		parameterCount:= pCurrentObject.getParametersCount();
		IF parameterCount>0 THEN
			FOR parameterIndex:=0 TO parameterCount-1 DO
				curData:=pCurrentObject.getParametrName(parameterIndex);
				SysFileStreamFPutS(File:=h_file,str:=ADR(devisor));
				SysFileStreamFPutS(File:=h_file,str:=ADR(curData));	
			END_FOR
		ELSE
				SysFileStreamFPutS(File:=h_file,str:=ADR(devisor));				
		END_IF			
		currentObject:=currentObject.NextElem;
	UNTIL 	currentObject =0
	END_REPEAT	
END_IF
END_METHOD

METHOD PRIVATE writeDataRow:BOOL
VAR_INPUT
		h_file:RTS_IEC_HANDLE;
		currentSlice:LAT.IElement;
END_VAR
VAR
	curData:STRING;
	currentObject: LAT.IElement;
	pCurrentObject:IObjectListener;	
	pCurrentSlice: POINTER TO TimeSlice;	
	parameterIndex:WORD;
	parameterCount:WORD;
END_VAR
__QUERYPOINTER (currentSlice,pCurrentSlice);
IF NOT pCurrentSlice^.values.ListIsEmpty THEN
	SysFileStreamFPutS(File:=h_file,str:=ADR(endln));
	curData:=timeToString(hrTime:=pCurrentSlice^.timeStamp);
	SysFileStreamFPutS(File:=h_file,str:=ADR(curData));

	currentObject:=pCurrentSlice^.values.HeadElem;
	REPEAT
		__QUERYINTERFACE (currentObject,pCurrentObject);

		parameterCount:= pCurrentObject.getParametersCount();
		IF parameterCount>0 THEN
			FOR parameterIndex:=0 TO parameterCount-1 DO
				curData:=pCurrentObject.getParametrValue(parameterIndex);
				SysFileStreamFPutS(File:=h_file,str:=ADR(devisor));
				SysFileStreamFPutS(File:=h_file,str:=ADR(curData));	
			END_FOR
		ELSE
				SysFileStreamFPutS(File:=h_file,str:=ADR(devisor));				
		END_IF		
		
		currentObject:=currentObject.NextElem;
	UNTIL 	currentObject =0
	END_REPEAT			
END_IF
writeDataRow:=pCurrentSlice^.timeStamp>=lastSavedTimeStamp;
END_METHOD

METHOD PRIVATE countinueDataWrite
VAR_INPUT
END_VAR
VAR
	timeKvant:TON:=(PT:=writeFileTimeKvant);
	isLastRow:BOOL;
END_VAR
timeKvant(IN:=FALSE);
timeKvant(IN:=TRUE);

IF currentWritedSlice=0 THEN
	currentWritedSlice:=TimeSlices.HeadElem;
END_IF;		
REPEAT
	isLastRow:= writeDataRow(archiveFileHandle,currentWritedSlice);
	timeKvant();
	currentWritedSlice:=currentWritedSlice.NextElem;
UNTIL 	(currentWritedSlice=0) OR isLastRow OR  timeKvant.Q
END_REPEAT	

IF isLastRow OR currentWritedSlice=0 THEN
	SysFileStreamFClose(File:=archiveFileHandle);
	archiveFileHandle:=0;
	currentWritedSlice:=0;
END_IF;
END_METHOD

METHOD PUBLIC register
VAR_INPUT
END_VAR
VAR

END_VAR
provider.RegisterArchive(nArchive:=THIS);
END_METHOD

METHOD FB_init : BOOL
VAR_INPUT
  bInitRetains : BOOL; // if TRUE, the retain variables are initialized (warm start / cold start)
  bInCopyCode : BOOL;  // if TRUE, the instance afterwards gets moved into the copy code (online change)
  table: POINTER TO TableDescriptor;
END_VAR
register();
END_METHOD

METHOD PUBLIC startAccident
VAR_INPUT
	descript:STRING;
END_VAR
IF NOT (accidentStarted OR (archiveFileHandle<>0)) THEN
	SysTimeRtcHighResGet(accidentTime);
	accidentStarted:=TRUE;	
	accidentDesc:=descript;
END_IF
END_METHOD

METHOD PUBLIC writeLog
VAR_INPUT
	fileName:STRING;
	append:BOOL;
END_VAR
VAR
	fileMode:STRING;
END_VAR
IF append THEN
	fileMode:='a';
ELSE
	fileMode:='w';		
END_IF
archiveFileHandle:=SysFileStreamFOpen(FileName:=fileName,Mode:=fileMode);

IF archiveFileHandle=0 THEN
	RETURN;
END_IF

IF lastTimeSlice<>0 THEN
	IF NOT append THEN
		writeHead(archiveFileHandle);
	END_IF
	countinueDataWrite();
ELSE
	SysFileStreamFClose(File:=archiveFileHandle);
	archiveFileHandle:=0;
END_IF
END_METHOD

END_FUNCTION_BLOCK

// lowLevel_ecl/EmergencyAarchive/TimeSlice
{attribute 'enable_dynamic_creation'}
FUNCTION_BLOCK INTERNAL TimeSlice EXTENDS LAT.Element
VAR_INPUT

END_VAR
VAR_OUTPUT
	values:LAT.List;
END_VAR
VAR
	_timeStamp:SYSTIME:=0;
END_VAR

METHOD PUBLIC appendValueListener
VAR_INPUT
	object:IObjectListener;
END_VAR
VAR
		newValueIterface: LAT.IElement;
END_VAR
IF object<>0 THEN
	IF (__QUERYINTERFACE(object,newValueIterface)) THEN
		values.AppendElem(newValueIterface);
	END_IF
END_IF
END_METHOD

METHOD PUBLIC copy : Pointer to TimeSlice
VAR_INPUT
END_VAR
VAR
	currentObject: LAT.IElement;
	pCurrentObject:IObjectListener;
	pNewObject:IObjectListener;
END_VAR
copy:=__NEW(TimeSlice);
IF copy<>0 THEN	
	IF NOT values.ListIsEmpty THEN
		currentObject:=values.HeadElem;
		REPEAT
			__QUERYINTERFACE (currentObject,pCurrentObject);
			pNewObject:=pCurrentObject.copy();
			IF pNewObject<>0 THEN
				copy^.appendValueListener(pNewObject);
				currentObject:=currentObject.NextElem;
			ELSE
				__DELETE(copy);
				currentObject:=0;
			END_IF
		UNTIL 	currentObject =0
		END_REPEAT
	END_IF
END_IF

IF copy=0 THEN
	LogAdd(CmpLog.STD_LOGGER,'EmergencyAarchive',UDINT_TO_DINT(CmpLog.LogClass.LOG_ERROR),0,0,'Not enough dynamic memory for new slice.');
END_IF
END_METHOD

METHOD PUBLIC update
VAR_INPUT
END_VAR
VAR
	currentObject: LAT.IElement;
	pCurrentObject:IObjectListener;
	tmpTimeStamp:SYSTIME:=0;
END_VAR
SysTimeRtcHighResGet(pTimestamp:= tmpTimeStamp);
timeStamp:= tmpTimeStamp;
IF NOT values.ListIsEmpty THEN
	currentObject:=values.HeadElem;
	REPEAT
		__QUERYINTERFACE (currentObject,pCurrentObject);
		pCurrentObject.update();
		currentObject:=currentObject.NextElem;
	UNTIL 	currentObject = 0
	END_REPEAT
END_IF
END_METHOD

PROPERTY PUBLIC timeStamp : SYSTIME
SET
_timeStamp:=timeStamp;
END_SET
GET
timeStamp:=_timeStamp;
END_GET
END_PROPERTY

METHOD FB_Exit : bool
VAR_INPUT
	bInCopyCode : BOOL; 
END_VAR
VAR
	currentObject: LAT.IElement;
	pCurrentObject:IObjectListener;
END_VAR
IF NOT values.ListIsEmpty THEN
	currentObject:=values.PopElem();
	REPEAT
		__QUERYINTERFACE (currentObject,pCurrentObject);
		deleteObjectListener(pCurrentObject);
		currentObject:=values.PopElem();
	UNTIL 	currentObject =0
	END_REPEAT
END_IF
END_METHOD

END_FUNCTION_BLOCK

// lowLevel_ecl/EmergencyAarchive/ObjectListener/IObjectListener
INTERFACE IObjectListener EXTENDS __SYSTEM.IQueryInterface

METHOD PUBLIC copy : IObjectListener
VAR_INPUT
END_VAR
END_METHOD

METHOD PUBLIC getName : String
VAR_INPUT
END_VAR
END_METHOD

METHOD update
VAR_INPUT
END_VAR
END_METHOD

METHOD getParametersCount : word
VAR_INPUT
END_VAR
END_METHOD

METHOD getParametrName : STRING
VAR_INPUT
	index:WORD;
END_VAR
END_METHOD

METHOD getParametrValue : String
VAR_INPUT
	index:WORD;
END_VAR
END_METHOD

END_INTERFACE

// lowLevel_ecl/EmergencyAarchive/ObjectListener/deleteObjectListener
FUNCTION INTERNAL deleteObjectListener : BOOL
VAR_INPUT
	object:IObjectListener;
END_VAR
VAR
	analogListener:POINTER TO AnalogObjectListener;
	discretListener:POINTER TO DiscretObjectListener;
	imListener:POINTER TO ImObjectListener;
END_VAR

//TODO: всегда вызывается __delete для discretListener. Как узнать сколько памяти освобождается?
IF __QUERYPOINTER(object,discretListener) THEN
	__DELETE(discretListener);
ELSIF __QUERYPOINTER(object,analogListener) THEN
	__DELETE(analogListener);
ELSIF __QUERYPOINTER(object,imListener) THEN
	__DELETE (imListener);
END_IF

END_FUNCTION

// lowLevel_ecl/EmergencyAarchive/ObjectListener/AnalogObjectListener
{attribute 'enable_dynamic_creation'}
FUNCTION_BLOCK INTERNAL FINAL AnalogObjectListener EXTENDS LAT.Element IMPLEMENTS IObjectListener
VAR_INPUT
	object: IAnalogArchObject;
END_VAR
VAR_OUTPUT
END_VAR
VAR
	value:REAL;
	srcValue:REAL;
	status: DWORD;
END_VAR

METHOD PUBLIC copy : IObjectListener
VAR_INPUT
END_VAR
VAR
	newIam:POINTER TO AnalogObjectListener;
END_VAR
newIam:=__NEW(AnalogObjectListener);
IF newIam<>0 THEN
	newIam^.object:=object;
	__QUERYINTERFACE(newIam^,copy);
END_IF
END_METHOD

METHOD PUBLIC getName : String
VAR_INPUT
END_VAR
getName:=object.archName;
END_METHOD

METHOD update
status:=object.archStatus;
value:=object.archValue;
srcValue:=object.archSrcValue;
END_METHOD

METHOD getParametersCount : WORD
getParametersCount:=3;
END_METHOD

METHOD getParametrName : STRING
VAR_INPUT
	index	: WORD;
END_VAR
CASE index OF
	0: getParametrName:='Status';
	1: getParametrName:='Value';
	2: getParametrName:='srcValue';
END_CASE
END_METHOD

METHOD getParametrValue : STRING
VAR_INPUT
	index	: WORD;
END_VAR
CASE index OF
	0: getParametrValue:=DWORD_TO_STRING(status);
	1: getParametrValue:=FPU.RealToStr(value);
	2: getParametrValue:=FPU.RealToStr(srcValue);
END_CASE
END_METHOD

END_FUNCTION_BLOCK

// lowLevel_ecl/EmergencyAarchive/ObjectListener/IAnalogArchObject
INTERFACE IAnalogArchObject EXTENDS IImArchObject

PROPERTY archValue : REAL
GET
END_GET
END_PROPERTY

PROPERTY archSrcValue : REAL
GET
END_GET
END_PROPERTY

END_INTERFACE

// lowLevel_ecl/EmergencyAarchive/ObjectListener/IImArchObject
INTERFACE IImArchObject EXTENDS IBaseArchObject

PROPERTY archStatus : DWORD
GET
END_GET
END_PROPERTY

END_INTERFACE

// lowLevel_ecl/EmergencyAarchive/ObjectListener/IBaseArchObject
INTERFACE IBaseArchObject EXTENDS __SYSTEM.IQueryInterface

PROPERTY archName : STRING
GET
END_GET
END_PROPERTY

END_INTERFACE

// lowLevel_ecl/EmergencyAarchive/ObjectListener/DiscretObjectListener
{attribute 'enable_dynamic_creation'}
FUNCTION_BLOCK INTERNAL FINAL DiscretObjectListener EXTENDS LAT.Element IMPLEMENTS IObjectListener
VAR_INPUT
	object: IDiscretArchObject;
END_VAR
VAR_OUTPUT
END_VAR
VAR
	value:WORD;
	reliability:WORD;
END_VAR

METHOD PUBLIC copy : IObjectListener
VAR_INPUT
END_VAR
VAR
	newIam:POINTER TO DiscretObjectListener;
END_VAR
newIam:=__NEW(DiscretObjectListener);
IF newIam<>0 THEN
	newIam^.object:=object;
	__QUERYINTERFACE(newIam^,copy);
END_IF;
END_METHOD

METHOD PUBLIC getName : String
VAR_INPUT
END_VAR
getName:=object.archName;
END_METHOD

METHOD update
value:=object.archValue;
reliability:=object.archReliability;
END_METHOD

METHOD getParametersCount : WORD
getParametersCount:=2;
END_METHOD

METHOD getParametrName : STRING
VAR_INPUT
	index	: WORD;
END_VAR
CASE index OF
	0: getParametrName:='Value';
	1: getParametrName:='Reliability';
END_CASE
END_METHOD

METHOD getParametrValue : STRING
VAR_INPUT
	index	: WORD;
END_VAR
CASE index OF
	0: getParametrValue:=WORD_TO_STRING(value);
	1: getParametrValue:=WORD_TO_STRING(reliability);
END_CASE
END_METHOD

END_FUNCTION_BLOCK

// lowLevel_ecl/EmergencyAarchive/ObjectListener/IDiscretArchObject
INTERFACE IDiscretArchObject EXTENDS IBaseArchObject

PROPERTY archValue : WORD
GET
END_GET
END_PROPERTY

PROPERTY archReliability : WORD
GET
END_GET
END_PROPERTY

END_INTERFACE

// lowLevel_ecl/EmergencyAarchive/ObjectListener/ImObjectListener
{attribute 'enable_dynamic_creation'}
FUNCTION_BLOCK INTERNAL FINAL ImObjectListener EXTENDS LAT.Element IMPLEMENTS IObjectListener
VAR_INPUT
	object: IImArchObject;
END_VAR
VAR_OUTPUT
END_VAR
VAR
	status: DWORD;
END_VAR

METHOD PUBLIC copy : IObjectListener
VAR_INPUT
END_VAR
VAR
	newIam:POINTER TO ImObjectListener;
END_VAR
newIam:=__NEW(ImObjectListener);
IF newIam<>0 THEN
	newIam^.object:=object;
	__QUERYINTERFACE(newIam^,copy);
END_IF
END_METHOD

METHOD PUBLIC getName : String
VAR_INPUT
END_VAR
getName:=object.archName;
END_METHOD

METHOD update
status:=object.archStatus;
END_METHOD

METHOD getParametersCount : WORD
getParametersCount:=1;
END_METHOD

METHOD getParametrValue : STRING
VAR_INPUT
	index	: WORD;
END_VAR
CASE index OF
	0: getParametrValue:=DWORD_TO_STRING(status);
END_CASE
END_METHOD

METHOD getParametrName : STRING
VAR_INPUT
	index	: WORD;
END_VAR
CASE index OF
	0: getParametrName:='Status';
END_CASE
END_METHOD

END_FUNCTION_BLOCK

// lowLevel_ecl/EmergencyAarchive/ObjectListener/createObjectListener
FUNCTION INTERNAL createObjectListener : BOOL
VAR_INPUT
	object: POINTER TO BaseObject;
END_VAR
VAR_OUTPUT
	newListener: IObjectListener;	
END_VAR
VAR
	iImObject:IImArchObject;	
	pImObject: POINTER TO ImObjectListener;
	
	iAnalogObject:IAnalogArchObject;	
	pAnalogObject: POINTER TO AnalogObjectListener;	
	
	iDiscretObject:IDiscretArchObject;	
	pDiscretObject: POINTER TO DiscretObjectListener;		
END_VAR

newListener:=0;
createObjectListener:=TRUE;

IF __QUERYINTERFACE(object^, iAnalogObject) THEN
	pAnalogObject:=__NEW(AnalogObjectListener);
	IF pAnalogObject<>0 THEN	
		pAnalogObject^.object:=iAnalogObject;
		__QUERYINTERFACE(pAnalogObject^,newListener);
	END_IF
ELSIF __QUERYINTERFACE(object^, iDiscretObject) THEN
	pDiscretObject:=__NEW(DiscretObjectListener);
	IF pDiscretObject <>0 THEN
		pDiscretObject^.object:=iDiscretObject;
		__QUERYINTERFACE(pDiscretObject^,newListener);
	END_IF
ELSIF __QUERYINTERFACE(object^, iImObject) THEN
	pImObject:=__NEW(ImObjectListener);
	IF pImObject <>0 THEN
		pImObject^.object:=iImObject;
		__QUERYINTERFACE(pImObject^,newListener);
	END_IF
ELSE
	createObjectListener:=FALSE;			
END_IF

END_FUNCTION

// lowLevel_ecl/kontroller/IKontroller
INTERFACE IKontroller

METHOD PUBLIC callCommands
VAR_INPUT
END_VAR
END_METHOD

METHOD PUBLIC callInputTable
VAR_INPUT
END_VAR
END_METHOD

METHOD callOutputTable
VAR_INPUT
END_VAR
END_METHOD

END_INTERFACE

// lowLevel_ecl/Common/fb/RP_trig
FUNCTION_BLOCK RP_trig
VAR_INPUT
	in:BOOL;
END_VAR
VAR_OUTPUT
	Qp:BOOL;
	Qn:BOOL;
END_VAR
VAR
	prtig:R_TRIG;
	ntrig:R_TRIG;
END_VAR

prtig(CLK:=in,Q=>Qp);
ntrig(CLK:= NOT in,Q=>Qn);

END_FUNCTION_BLOCK

// lowLevel_ecl/Common/table/callExec
FUNCTION callExec : BOOL
VAR_INPUT
	CONSTANT table:TableDescriptor;
END_VAR
VAR
	curObject:POINTER TO BaseObject;
END_VAR

curObject:=table.head;
IF curObject=0 THEN
	RETURN;
END_IF
REPEAT
	callObject(curObject);
	curObject:=curObject^.getNext();
	UNTIL curObject=0
END_REPEAT

END_FUNCTION

// lowLevel_ecl/Common/table/callObject
FUNCTION callObject : bool
VAR_INPUT
	object:POINTER TO BaseObject;
END_VAR
VAR
	IcurIm:ObjectCommands;
END_VAR

object^();
IF (__QUERYINTERFACE(object^,IcurIm)) THEN
	IcurIm.writeImStatus();
END_IF

END_FUNCTION

// lowLevel_ecl/im/BaseIms/ObjectCommands
INTERFACE ObjectCommands EXTENDS __SYSTEM.IQueryInterface

METHOD PUBLIC DisableOpcControl
VAR_INPUT
END_VAR
END_METHOD

METHOD FINAL execCommand
VAR_INPUT
END_VAR
END_METHOD

PROPERTY hasCommand : Bool
GET
END_GET
END_PROPERTY

METHOD EnableOpcControl
VAR_INPUT
END_VAR
END_METHOD

METHOD PUBLIC writeImStatus
VAR_INPUT
END_VAR
END_METHOD

END_INTERFACE

// lowLevel_ecl/kontroller/baseSources/ISource
INTERFACE ISource

PROPERTY imit : bool
GET
END_GET
SET
END_SET
END_PROPERTY

END_INTERFACE

// lowLevel_ecl/algoritms/ExecComands
FUNCTION ExecComands : BOOL
VAR_INPUT
	table:TableDescriptor;
END_VAR
VAR
		curObject:POINTER TO BaseObject;
		IcurIm:ObjectCommands;
END_VAR

curObject:=table.head;
IF curObject<>0 THEN
	REPEAT
		IF (__QUERYINTERFACE(curObject^,IcurIm)) THEN		
			IcurIm.execCommand();
		END_IF;
		curObject:=curObject^.getNext();
	UNTIL curObject=0
	END_REPEAT;
END_IF;

END_FUNCTION

// lowLevel_ecl/kontroller/mlp/Diagnostic/DiagnosticMlp
{attribute 'symbol' := 'none'}
FUNCTION_BLOCK PUBLIC DiagnosticMlp
VAR_INPUT
	elpk:POINTER TO Elpk04;
	bsStatusBaseAdress:INT:=64;
END_VAR
VAR_OUTPUT
	{attribute 'symbol' := 'read'}
	Config:STRING(2048);
	{attribute 'symbol' := 'read'}
	Status:STRING(4096);

	BsConf:ARRAY[1..8]OF BsDescriptor;
	BsStatus:ARRAY[1..8] OF BsStatusDecriptor;
	
	ns:BOOL;
END_VAR
VAR
	confFile:iniFileReader;
	
	mlpConnect:TOF:=(PT:=T#2S);
	mlpLastCounter:WORD;
	
	init:BOOL;
	bsStatusIndexses:ARRAY[1..8] OF INT;
	
	{attribute 'symbol' := 'read'}
	link:INT;
	linkGen:GEN;
END_VAR
VAR_TEMP
	bsIndex:INT;
	i:INT;
END_VAR
VAR CONSTANT
	mlpLifeCounter:INT:=63;	
END_VAR

IF NOT init THEN
	FOR i:=1 TO 8 DO
		bsStatusIndexses[i]:=bsStatusBaseAdress+(i-1);
	END_FOR 
	init:=TRUE;
END_IF

mlpConnect(IN:=elpk^.DIn_[mlpLifeCounter].val<>mlpLastCounter);
mlpLastCounter:=elpk^.DIn_[mlpLifeCounter].val;

ns:=FALSE;

FOR bsIndex:=1 TO 8 DO
	IF BsConf[bsIndex].enabled THEN
		BsStatus[bsIndex].connected:= elpk^.DIn_[bsStatusIndexses[bsIndex]].val=7;
		ReadModules(bsConnected:=BsStatus[bsIndex].connected AND mlpConnect.Q,bsIndex:=bsIndex);
	END_IF
END_FOR

writeStatus();

linkGen(MODE:=TRIANGLE,AMPLITUDE:=32767,CYCLES:=32767,BASE:=FALSE,OUT=>link);

METHOD PRIVATE WriteConfig
VAR_INPUT
END_VAR
VAR
	source:PT_SIZE;
	dest:PT_SIZE;
	result:BYTE;
	i:UINT;
	curByte:POINTER TO BYTE;
END_VAR
source.pString:=ADR(BsConf);
source.uiSize:=SIZEOF(BsConf);
dest:=BASE64(TextToEncode:=source,isLastBlock:=TRUE,pbyError:=ADR(result));
FOR i:=0 TO dest.uiSize-1 DO
	curByte:=dest.pString+i;
	Config[i]:=curByte^;	
END_FOR
END_METHOD

METHOD PUBLIC writeStatus
VAR_INPUT
	
END_VAR
VAR
	source:PT_SIZE;
	dest:PT_SIZE;
	result:BYTE;
	i:UINT;
	curByte:POINTER TO BYTE;
END_VAR
source.pString:=ADR(BsStatus);
source.uiSize:=SIZEOF(BsStatus);
dest:=BASE64(TextToEncode:=source,isLastBlock:=TRUE,pbyError:=ADR(result));
FOR i:=0 TO dest.uiSize-1 DO
	curByte:=dest.pString+i;
	Status[i]:=curByte^;	
END_FOR
END_METHOD

METHOD PRIVATE ReadModules
VAR_INPUT
	bsConnected:BOOL;
	bsIndex:INT;
END_VAR
VAR
		moduleIndex:INT;
END_VAR
FOR moduleIndex:=1 TO 15 DO
	IF BsConf[bsIndex].modules[moduleIndex].moduleType<>0 THEN
		IF bsConnected THEN
			BsStatus[bsIndex].modules[moduleIndex].moduleStatus.0:=NOT FaultModel(mIndex:= BsConf[bsIndex].modules[moduleIndex].addr,TypeModule:= BsConf[bsIndex].modules[moduleIndex].moduleType,FirstNomComPort:=0);
			
			//IF 	BsStatus[bsIndex].modules[moduleIndex].moduleStatus.0=TRUE THEN
				CASE BsConf[bsIndex].modules[moduleIndex].moduleType OF
					ModuleTypes.DI8:
						readDi8Status(bs:=bsIndex,module:=moduleIndex);
					ModuleTypes.AI4:
						readAI4Status(bs:=bsIndex,module:=moduleIndex);
					ModuleTypes.OA4:
						readOA4Status(bs:=bsIndex,module:=moduleIndex);
				END_CASE
			//END_IF
			IF NOT BsStatus[bsIndex].modules[moduleIndex].moduleStatus.0 THEN
				ns:=TRUE;
			END_IF
		ELSE
			BsStatus[bsIndex].modules[moduleIndex].moduleStatus:=0;
			ns:=TRUE;
		END_IF;
	END_IF
END_FOR
END_METHOD

METHOD PRIVATE FaultModel : BOOL
VAR_INPUT
//	DataM: DiagnosticIndex; // Данные для вычисления индекса битовой пары в массиве ERR 
	mIndex: WORD; // Индекс первого канала в MLP модуля УСО
	TypeModule: ModuleTypes; // Тип модуля УСО
	FirstNomComPort: WORD; // Первый номер COM порта модуля RS485 
END_VAR
VAR
	Index: WORD; // Индекс в массиве ERR
	NomTwoBits: WORD; // Номер битовой пары
END_VAR
FaultModel := FALSE;
IF TypeModule <> ModuleTypes.none THEN
	CASE TypeModule OF	
		ModuleTypes.DI8, ModuleTypes.RS485:
			Index := mIndex / 8;
			NomTwoBits := mIndex - (Index * 8); 	
		ModuleTypes.DO5, ModuleTypes.IF3:
			Index := 16 +mIndex / 8;
			NomTwoBits := mIndex - (mIndex / 8) * 8;
		ModuleTypes.AI4:
			Index := 32 + ((mIndex / 4)/ 8);
			NomTwoBits := (mIndex / 4) MOD 8;
		ModuleTypes.OA4:
			Index := 48 + ((mIndex / 4)/ 8);
			NomTwoBits := (mIndex / 4) MOD 8;
	END_CASE	
	
	CASE NomTwoBits OF
		0:
			IF elpk^.Diag_[Index].0 OR  elpk^.Diag_[Index].1 THEN
				FaultModel := TRUE;
			END_IF
		1:
			IF elpk^.Diag_[Index].2 OR  elpk^.Diag_[Index].3 THEN
				FaultModel := TRUE;
			END_IF
		2:
			IF elpk^.Diag_[Index].4 OR  elpk^.Diag_[Index].5 THEN
				FaultModel := TRUE;
			END_IF
		3:
			IF elpk^.Diag_[Index].6 OR  elpk^.Diag_[Index].7 THEN
				FaultModel := TRUE;
			END_IF
		4:
			IF elpk^.Diag_[Index].8 OR  elpk^.Diag_[Index].9 THEN
				FaultModel := TRUE;
			END_IF
		5:
			IF elpk^.Diag_[Index].10 OR  elpk^.Diag_[Index].11 THEN
				FaultModel := TRUE;
			END_IF
		6:
			IF elpk^.Diag_[Index].12 OR  elpk^.Diag_[Index].13 THEN
				FaultModel := TRUE;
			END_IF
		7:
			IF elpk^.Diag_[Index].14 OR  elpk^.Diag_[Index].15 THEN
				FaultModel := TRUE;
			END_IF				
	END_CASE
	IF TypeModule = ModuleTypes.RS485 AND (elpk^.DIn_[mIndex].val = 0 (*OR elpk^.DIn_[mIndex].val <> FirstNomComPort*)) THEN		
		FaultModel := TRUE;	
	END_IF
END_IF
END_METHOD

METHOD PRIVATE readDi8Status
VAR_INPUT
	bs: INT;
	module:INT;
END_VAR
BsStatus[bs].modules[module].pinStatus:=elpk^.DIn_[BsConf[bs].modules[module].addr].val;
IF (elpk^.DIn_[BsConf[bs].modules[module].addr].val AND 16#AAAA)<>16#AAAA THEN
	ns:=TRUE;
END_IF
END_METHOD

METHOD PRIVATE readAI4Status
VAR_INPUT
	bs: INT;
	module:INT;
END_VAR
VAR
	pinStatus:smartWordPack;
	channel:word;
END_VAR
pinStatus(status:= BsStatus[bs].modules[module].pinStatus);
FOR channel:=0 TO 3 DO
	pinStatus.setBits(start:=channel*2,end:=channel*2,value:=BOOL_TO_WORD(elpk^.AIn_[BsConf[bs].modules[module].addr+channel].f.4 OR elpk^.AIn_[BsConf[bs].modules[module].addr+channel].f.5));
	pinStatus.setBits(start:=channel*2+1,end:=channel*2+1,value:=BOOL_TO_WORD(elpk^.AIn_[BsConf[bs].modules[module].addr+channel].f.2));
	IF NOT elpk^.AIn_[BsConf[bs].modules[module].addr+channel].f.2 THEN
		ns:=TRUE;
	END_IF
END_FOR
END_METHOD

METHOD PRIVATE readOA4Status
VAR_INPUT
	bs: INT;
	module:INT;
END_VAR
VAR
	pinStatus:smartWordPack;
	channel:word;
END_VAR
pinStatus(status:= BsStatus[bs].modules[module].pinStatus);
FOR channel:=0 TO 3 DO
	pinStatus.setBits(start:=channel*2,end:=channel*2+1,value:=2);
END_FOR
END_METHOD

METHOD PUBLIC readConfig
VAR_INPUT
	mlpConfig:STRING;
END_VAR
VAR
	iba:INT;
	currentLine:iniFileLine;
	
	bs:WORD;
	module:WORD;
	
	_bsPos:INT;
	_modPos:INT;
	isModuleSection:BOOL;
	i:INT;
	
END_VAR
IF NOT confFile.open(configFile:=mlpConfig)THEN
	return;
END_IF

currentLine:=confFile.readLn();
WHILE currentLine.status<>iniFileStatus.Eof DO
	CASE(currentLine.status) OF
		iniFileStatus.Section:
			_bsPos:=FIND(STR1:=currentLine.Section,STR2:='T');
			_modPos:=FIND(STR1:=currentLine.Section,STR2:='_X');
			IF (_bsPos<>0) AND (_modPos<>0) THEN
				bs:=STRING_TO_WORD(MID(STR:=currentLine.Section,POS:=_bsPos+1,LEN:=_modPos-_bsPos));
				module:=STRING_TO_WORD(RIGHT(STR:=currentLine.Section,SIZE:=LEN(STR:=currentLine.Section)-_modPos-1));
				IF ((bs>0) AND (module>0) )	THEN			
					isModuleSection:=TRUE;
					BsConf[bs].enabled:=TRUE;
				END_IF
			ELSE
				isModuleSection:=FALSE;
			END_IF
			
		iniFileStatus.Parametr:
			IF isModuleSection THEN				
				IF (currentLine.Parameter='CH_IN') OR (currentLine.Parameter='CH_OUT') THEN
					BsConf[bs].modules[module].addr:=STRING_TO_WORD(currentLine.Value);
				ELSIF currentLine.Parameter='MOD' THEN
					BsConf[bs].modules[module].moduleType:=HexString_to_Word(currentLine.Value);
				ELSIF currentLine.Parameter='FUNC' THEN
					BsConf[bs].modules[module].funct:=STRING_TO_BYTE(currentLine.Value);						
				END_IF
			END_IF
	END_CASE
	currentLine:=confFile.readLn();
END_WHILE

confFile.close();

WriteConfig();
END_METHOD

METHOD PUBLIC readConfig_faleev
VAR_INPUT
	mlpConfig:STRING;
END_VAR
VAR
	iba:INT;
	currentLine:iniFileLine;
	
	bs:WORD;
	module:WORD;
	
	_bsPos:INT;
	_modPos:INT;
	isModuleSection:BOOL;
	i:INT;
	
END_VAR
//	0x00=NONE - нет никакого модуля
//	0x01 (MODTYPE_AIN8)		= МАЦП-03-08
//	0x11 (MODTYPE_AIN16)	= МАЦП-03-16
//	0x02 (MODTYPE_DIN)		= МПЦ-03-16
//	0x03 (MODTYPE_DOUT)		= МТЦ-03-16
//	0x04 (MODTYPE_DAC4)		= МЦАП-03-04
//	0x82 (MODTYPE_MXDIN)	= МПЦ-03-16 MX
//	0x83 (MODTYPE_MXDOUT)	= МТЦ-03-16 MX

	// BsConf[1..8]			modules[1..16]
	BsConf[1].enabled:=TRUE;
	BsConf[1].modules[1].moduleType:= 16#82;	// MOD = MXDIN
	BsConf[1].modules[1].addr:= 0;				// CH_IN	- начиная с DIN0...
	BsConf[1].modules[1].funct:= 2;			// Func	- ввод

	BsConf[1].modules[2].moduleType:= 16#03;	// MOD = DOUT16
	BsConf[1].modules[2].addr:= 2;				// CH_OUT	- DOUT2
	BsConf[1].modules[2].funct:= 1;			// Func	- вывод
	
	BsConf[1].modules[3].moduleType:= 16#83;	// MOD = MXDOUT
	BsConf[1].modules[3].addr:= 0;				// CH_OUT	- не используется
	BsConf[1].modules[3].funct:= 1;			// Func	- вывод
		
	BsConf[1].modules[4].moduleType:= 16#03;	// MOD = DOUT16
	BsConf[1].modules[4].addr:= 3;				// CH_OUT	- DOUT3
	BsConf[1].modules[4].funct:= 1;			// Func	- вывод
	
	BsConf[1].modules[5].moduleType:= 16#03;			// MOD = DOUT16
	BsConf[1].modules[5].addr:= 0;					// CH_OUT	- DOUT0
	BsConf[1].modules[5].funct:= 1;					// Func	- вывод
	
	BsConf[1].modules[6].moduleType:= 16#03;	// MOD = DOUT16
	BsConf[1].modules[6].addr:= 4;				// CH_OUT	- DOUT4
	BsConf[1].modules[6].funct:= 1;				// Func	- вывод
	
	BsConf[1].modules[7].moduleType:= 16#03;	// MOD = DOUT16
	BsConf[1].modules[7].addr:= 1;				// CH_OUT	- DOUT1
	BsConf[1].modules[7].funct:= 1;				// Func	- вывод
	
	BsConf[1].modules[8].moduleType:= 16#02;	// MOD = DIN16
	BsConf[1].modules[8].addr:= 14;				// CH_IN	- DOUT14
	BsConf[1].modules[8].funct:= 2;				// Func	- ввод

	BsConf[1].modules[9].moduleType:= 16#01;	// MOD = AIN8
	BsConf[1].modules[9].addr:= 0;				// CH_IN	- AIN0..7
	BsConf[1].modules[9].funct:= 2;				// Func	- ввод

	BsConf[1].modules[10].moduleType:= 16#00;	// MOD = none
	BsConf[1].modules[10].addr:= 0;				// CH_IN
	BsConf[1].modules[10].funct:= 0;			// Func

	BsConf[1].modules[11].moduleType:= 16#01;	// MOD = AIN8
	BsConf[1].modules[11].addr:= 8;				// CH_IN	- AIN8..15
	BsConf[1].modules[11].funct:= 2;			// Func	- ввод

	BsConf[1].modules[12].moduleType:= 16#00;	// MOD = none
	BsConf[1].modules[12].addr:= 0;				// CH_IN
	BsConf[1].modules[12].funct:= 0;			// Func

	BsConf[1].modules[13].moduleType:= 16#01;	// MOD = AIN8
	BsConf[1].modules[13].addr:= 16;			// CH_IN	- AIN16..23
	BsConf[1].modules[13].funct:= 2;			// Func	- ввод

	BsConf[1].modules[14].moduleType:= 16#00;	// MOD = none
	BsConf[1].modules[14].addr:= 0;				// CH_IN
	BsConf[1].modules[14].funct:= 0;			// Func
	
	BsConf[1].modules[15].moduleType:= 16#01;	// MOD = AIN8
	BsConf[1].modules[15].addr:= 24;			// CH_IN	- AIN24..31
	BsConf[1].modules[15].funct:= 2;			// Func	- ввод

	BsConf[1].modules[16].moduleType:= 16#03;	// MOD = DOUT16
	BsConf[1].modules[16].addr:= 5;				// CH_OUT	- DOUT5
	BsConf[1].modules[16].funct:= 1;			// Func	- вывод





WriteConfig();
END_METHOD

END_FUNCTION_BLOCK

// lowLevel_ecl/kontroller/mlp/Diagnostic/iniFile/iniFileReader
{attribute 'symbol' := 'none'}
FUNCTION_BLOCK PUBLIC iniFileReader
VAR_INPUT	
END_VAR
VAR_OUTPUT
END_VAR
VAR
	fileHandle:RTS_IEC_HANDLE;
	lastSection:STRING;
END_VAR

METHOD PUBLIC open : BOOL
VAR_INPUT
	configFile:STRING;
END_VAR
VAR
	result:RTS_IEC_RESULT;
END_VAR

fileHandle:=SysFileStreamFOpen(FileName:=configFile,Mode:='r');
open:= fileHandle<>0;
END_METHOD

METHOD PUBLIC close
VAR_INPUT
END_VAR
SysFileStreamFClose(File:=fileHandle);
END_METHOD

METHOD PUBLIC readLn : iniFileLine
VAR_INPUT
END_VAR
VAR
	line:STRING;
	sectionStart:INT;
	parametrDevider:INT;
	garbagePos:INT;
END_VAR
REPEAT	
	IF SysFileStreamFGetS(File:=fileHandle,n:=SIZEOF(line),str:=ADR(line)) <> 0 THEN
	
		garbagePos:=FIND(STR1:=line,STR2:='$N');
		IF garbagePos<>0 THEN
			line:=DELETE(STR:=line,POS:=garbagePos,LEN:=2);
		END_IF
	
		sectionStart:=FIND(STR1:=line,STR2:='[');
		IF sectionStart<>0 THEN
			line:=DELETE(STR:=line,LEN:=1,POS:=sectionStart);
			line:=DELETE(STR:=line,LEN:=1,POS:=FIND(STR1:=line,STR2:=']'));
			lastSection:=line;
			readLn.Parameter:='';
			readLn.Value:='';
			readLn.status:=iniFileStatus.Section;
		ELSE
			parametrDevider:=FIND(STR1:=line,STR2:='=');
			IF parametrDevider<>0 THEN
				readLn.Parameter:=LEFT(STR:=line,SIZE:=parametrDevider-1);
				readLn.Value:=RIGHT(STR:=line,SIZE:=LEN(STR:=line)-parametrDevider);
				readLn.status:=iniFileStatus.Parametr;			
			END_IF	
		END_IF
	
		readLn.Section:=lastSection;
	ELSE
		readLn.status:=iniFileStatus.Eof;		
	END_IF;
UNTIL readLn.status<>iniFileStatus.NotDefined
END_REPEAT
END_METHOD

END_FUNCTION_BLOCK

// lowLevel_ecl/Common/smartPack/smartWordPack
	{attribute 'symbol' := 'none'}
	{attribute 'reflection'}
FUNCTION_BLOCK smartWordPack//Упаковывает биты в двойное слово. 
(*Выдает ошибку в журнал если полсе reset() записывались одни и теже биты.
*)
VAR_INPUT	
	status:REFERENCE TO WORD;//указатель на двойное слово
END_VAR
VAR_OUTPUT
END_VAR
VAR
	settedBits:DWORD;
	bitsAlredySetted:AloneLogMessage;
	bitsOutOfRenge:AloneLogMessage;
	{attribute 'instance-path'} 
	{attribute 'noinit'} 
	name: STRING; 
END_VAR
VAR CONSTANT

END_VAR

METHOD PUBLIC reset //сброс контроля перезаписи
VAR_INPUT
END_VAR
settedBits:=0;
END_METHOD

METHOD setBit 
//установить 1 бит
VAR_INPUT
	bitNum:WORD;// номер бита (с 0)
	value:BOOL;//Значение бита
END_VAR
setBits(bitNum,bitNum,bool_to_word(value));
END_METHOD

METHOD PUBLIC setBits //Устанавливает последовательность бит
VAR_INPUT
	start:WORD;//номер первого бита(с 0) 
	end:word;//номер последнего бита(с 0)
	value:WORD;//значение. Записывается start-end+1 младших бит.
END_VAR
VAR
	statusMask:WORD;
	bitsCount:WORD;
END_VAR
IF (start<0) OR (start>15) OR (end<0) OR (end>15) OR (start>end) THEN
	bitsOutOfRenge.write(CmpLog.LogClass.LOG_ERROR,name,'Nums out of range: ');	
	RETURN;
END_IF

bitsCount:=end-start+1;
statusMask:=SHL(SHL(1,bitsCount)-1,start);
IF (settedBits AND statusMask)<>0 THEN
	bitsAlredySetted.write(CmpLog.LogClass.LOG_ERROR,name,'Conflict bits: ');
END_IF
settedBits:=settedBits OR statusMask;
status:=(status AND NOT statusMask) OR (SHL(value,start) AND statusMask);
END_METHOD

END_FUNCTION_BLOCK

// lowLevel_ecl/Common/AloneLogMessage
FUNCTION_BLOCK AloneLogMessage
VAR_INPUT
END_VAR
VAR_OUTPUT
END_VAR
VAR
	writed:BOOL;
END_VAR

METHOD write
VAR_INPUT
	logClass:UDINT;
	name:STRING;
	message:STRING;
END_VAR
IF NOT writed THEN
	LogAdd(CmpLog.STD_LOGGER,name,UDINT_TO_DINT(logClass),0,0,CONCAT(message,name));
	writed:=true;
END_IF;
END_METHOD

END_FUNCTION_BLOCK

// lowLevel_ecl/Common/functions/HexString_to_Word
FUNCTION HexString_to_Word : WORD
VAR_INPUT
	hexValue:STRING;
END_VAR
VAR
	startPos:INT;
	lByteS:STRING(2);
	hByteS:STRING(2);
	lByte:WORD;
	hByte:WORD;
END_VAR

IF (LEFT(STR:=hexValue,SIZE:=2)='0x') THEN
	HByteS:=MID(STR:=hexValue,POS:=3,LEN:=2);
	lByteS:=MID(STR:=hexValue,POS:=5,LEN:=2);
	
	hByte:=SHL(BYTE_TO_WORD(hByteS[0]),8) OR BYTE_TO_WORD(hByteS[1]);
	lByte:=SHL(BYTE_TO_WORD(lByteS[0]),8) OR BYTE_TO_WORD(lByteS[1]);
	
	HexString_to_Word:=SHL(BYTE_TO_WORD(HEXinASCII_TO_BYTE(W:=hByte)),8) OR BYTE_TO_WORD(HEXinASCII_TO_BYTE(W:=lByte));
END_IF

END_FUNCTION

// lowLevel_ecl/kontroller/mlp/Sources/IMlpSource
INTERFACE IMlpSource EXTENDS __SYSTEM.IQueryInterface

METHOD setKontroller
VAR_INPUT
	nKontroller:REFERENCE TO Elpk04;
END_VAR
END_METHOD

END_INTERFACE

// K1/std12k5/Elpk_03_02/MainUP_PRG
PROGRAM MainUP_PRG
VAR
	START_INDEX, INDEX, INDEX2:INT:=0;
	
	I1,I2,I3,I4,I5,I6:INT;
	J1,J2,J3,J4,J5,J6,J7,J8,J9:INT;
	WWW1, WWW2, WWW3, WWW4, WWW5, WWW6, WWW7, WWW8:WORD;
	//ERR1, ERR2, ERR3, ERR4, ERR5, ERR6, ERR7, ERR8, ERR9, ERR22:RTS_IEC_RESULT;
	//ERR101, ERR102, ERR103, ERR104, ERR105,  ERR122:RTS_IEC_RESULT;
	//szFile1,szFile2:REFERENCE TO STRING;
	WW_WW1, WW_WW2, WW_WW3, WW_WW4:WORD;
	

//	GEN1:GEN;
//	IGEN1:INT;
/////////////////////////////////////////////////////////////////////////////////////////////////////////////
   {attribute 'displaymode':='hex'}
	MxStatus:WORD;		// OPC
//   {attribute 'displaymode':='hex'}
//	MxStatus_I:WORD;		// внутреннее использование

   {attribute 'displaymode':='hex'}
	MxMode:WORD;		// MX Active = 8
   {attribute 'displaymode':='hex'}
	//MxMode_O:WORD;		// внутреннее использование

	ADCWAY_I:WORD;
	ADCWAY_II:WORD;		// внутреннее использование
	
	ADCWAY_O:WORD;
	ADCWAY_OO:WORD;		// внутреннее использование

   {attribute 'displaymode':='hex'}
	BMPPRES:WORD;		// OPC
//   {attribute 'displaymode':='hex'}
//	BMPPRES_I:WORD;		// внутреннее использование

   {attribute 'displaymode':='hex'}
	BMPERR:WORD;		// OPC
///   {attribute 'displaymode':='hex'}
///	BMPERR_I:WORD;		// внутреннее использование

	MXLINES_I:WORD;
	MXLINES:WORD;
	
	HIDE_ERR_OUT_I:WORD;
	HIDE_ERR_OUT_II:WORD;

	HIDE_ERR_OUT_O:WORD;
	HIDE_ERR_OUT_OO:WORD;
	RWH_PERIOD_I:WORD;
	RWH_PERIOD:WORD;

	MX_ATT_I:WORD;
	MX_ATT:WORD;

	EXTCMD_I:WORD;
	EXTCMD:WORD;
   {attribute 'displaymode':='hex'}
	WDOG_O:WORD;
	
	
	
	
	// для отладки
   {attribute 'displaymode':='hex'}
	CH_MODCONF:WORD;
   {attribute 'displaymode':='hex'}
	CH_ERRNOW:WORD;
   {attribute 'displaymode':='hex'}
	CH_ERRHIST:WORD;
   {attribute 'displaymode':='hex'}
	CH_NDIAG:WORD;
   {attribute 'displaymode':='hex'}
	CH_MDIAG:WORD;
   {attribute 'displaymode':='hex'}
	CH_FIRMVER:WORD;
   {attribute 'displaymode':='hex'}
	CH_FIRMDATE:WORD;
   {attribute 'displaymode':='hex'}
	CH_CH7:WORD;
	// конец для отладки
(*
	MODULE_01:T_DIAGNOSTIC;
	MODULE_02:T_DIAGNOSTIC;
	MODULE_03:T_DIAGNOSTIC;
	MODULE_04:T_DIAGNOSTIC;
	MODULE_05:T_DIAGNOSTIC;
	MODULE_06:T_DIAGNOSTIC;
	MODULE_07:T_DIAGNOSTIC;
	MODULE_08:T_DIAGNOSTIC;
	MODULE_09:T_DIAGNOSTIC;
	MODULE_10:T_DIAGNOSTIC;
	MODULE_11:T_DIAGNOSTIC;
	MODULE_12:T_DIAGNOSTIC;
	MODULE_13:T_DIAGNOSTIC;
	MODULE_14:T_DIAGNOSTIC;
	MODULE_15:T_DIAGNOSTIC;
	MODULE_16:T_DIAGNOSTIC;
	*)

(*
   {attribute 'displaymode':='hex'}
	NodeErr1:WORD;	// OPC		
	///NodeErr1_Log:AddLOG_W_UP;// FB для записи NodeErr в лог при изменении значения	
   {attribute 'displaymode':='hex'}
	NodeErr2:WORD;	// OPC	
	///NodeErr2_Log:AddLOG_W_UP;// FB для записи NodeErr в лог при изменении значения	
   {attribute 'displaymode':='hex'}
	NodeErr3:WORD;	// OPC	
	///NodeErr3_Log:AddLOG_W_UP;// FB для записи NodeErr в лог при изменении значения	
   {attribute 'displaymode':='hex'}
	NodeErr4:WORD;	// OPC	
	///NodeErr4_Log:AddLOG_W_UP;// FB для записи NodeErr в лог при изменении значения	
   {attribute 'displaymode':='hex'}
	NodeErr5:WORD;	// OPC	
	///NodeErr5_Log:AddLOG_W_UP;// FB для записи NodeErr в лог при изменении значения	
   {attribute 'displaymode':='hex'}
	NodeErr6:WORD;	// OPC	
	///NodeErr6_Log:AddLOG_W_UP;// FB для записи NodeErr в лог при изменении значения	
   {attribute 'displaymode':='hex'}
	NodeErr7:WORD;	// OPC	
	///NodeErr7_Log:AddLOG_W_UP;// FB для записи NodeErr в лог при изменении значения	
   {attribute 'displaymode':='hex'}
	NodeErr8:WORD;	// OPC	
	///NodeErr8_Log:AddLOG_W_UP;// FB для записи NodeErr в лог при изменении значения	
   {attribute 'displaymode':='hex'}
	NodeErr9:WORD;	// OPC	
	///NodeErr9_Log:AddLOG_W_UP;// FB для записи NodeErr в лог при изменении значения	
   {attribute 'displaymode':='hex'}
	NodeErr10:WORD;	// OPC
	///NodeErr10_Log:AddLOG_W_UP;// FB для записи NodeErr в лог при изменении значения	
   {attribute 'displaymode':='hex'}
	NodeErr11:WORD;	// OPC
	///NodeErr11_Log:AddLOG_W_UP;// FB для записи NodeErr в лог при изменении значения	
   {attribute 'displaymode':='hex'}
	NodeErr12:WORD;	// OPC
	///NodeErr12_Log:AddLOG_W_UP;// FB для записи NodeErr в лог при изменении значения	
   {attribute 'displaymode':='hex'}
	NodeErr13:WORD;	// OPC
	///NodeErr13_Log:AddLOG_W_UP;// FB для записи NodeErr в лог при изменении значения	
   {attribute 'displaymode':='hex'}
	NodeErr14:WORD;	// OPC
	///NodeErr14_Log:AddLOG_W_UP;// FB для записи NodeErr в лог при изменении значения	
   {attribute 'displaymode':='hex'}
	NodeErr15:WORD;	// OPC
	///NodeErr15_Log:AddLOG_W_UP;// FB для записи NodeErr в лог при изменении значения	
   {attribute 'displaymode':='hex'}
	NodeErr16:WORD;	// OPC
	///NodeErr16_Log:AddLOG_W_UP;// FB для записи NodeErr в лог при изменении значения	

	///ImitatorON_Log:AddLOG_W_UP;// FB для записи в лог при изменении значения	

*)
END_VAR

// только для тестирования !!!
(*od.do_1.bits[0]:=0;*)
(*od.do_1.bits[1]:=1;
od.do_1.bits[2]:=1;
od.do_1.bits[3]:=1;
od.do_1.bits[4]:=1;
od.do_1.bits[5]:=1;
od.do_1.bits[6]:=1;
od.do_1.bits[7]:=1;

od.do_1.bits[8]:=1;
od.do_1.bits[9]:=1;
od.do_1.bits[10]:=1;
od.do_1.bits[11]:=1;
od.do_1.bits[12]:=1;
od.do_1.bits[13]:=1;
od.do_1.bits[14]:=1;
od.do_1.bits[15]:=1;
*)






	//
	// Формирование пилы жизни для передачи в ОРС. Значения от 0 до 1023. На каждом цикле +1.
	//
	LifeCnt:= (LifeCnt+1)AND 16#3FF;


///////////////////////////////////////////////////////////////////////////////////////////////////
//	Читать диагностику

	MxStatus:=MxStatus_I;	// OPC

	ADCWAY_II:=ADCWAY_I;
	BMPPRES_K:= BMPPRES:= BMPPRES_I;// в ОРС


	(*IF Imitator_code=16#55AA
	THEN// если есть имитатор - брать диагностику из имитатора и передать а ОРС
		BMPERR:=BMPERR_UP1_Im;// в ОРС
	ELSE
	// нет имитатора - брать диагностику из драйвера и передать в ОРС
		BMPERR:=BMPERR_I;// в ОРС
	END_IF
	BMPERR_K:=	BMPERR;*)
	BMPERR_K:=	BMPERR:=	BMPERR_I;// в ОРС

		
	MXLINES:=MXLINES_I;
	HIDE_ERR_OUT_II:=HIDE_ERR_OUT_I;
	RWH_PERIOD:=RWH_PERIOD_I;
	MX_ATT:=MX_ATT_I;
	EXTCMD:=EXTCMD_I;
	
//	ADCWAY_O:=%QW2;
//	HIDE_ERR_OUT_O:=%QW9;
//	WDOG_O:=16#55AA;	// Включить watchdog



	MasterOPC_ST:=REZERV1.MasterOPC;
	
	
	NodeErr1_K:= 	MODULES03[1].CH_NDIAG;
	NodeErr2_K:= 	MODULES03[2].CH_NDIAG;
	NodeErr3_K:= 	MODULES03[3].CH_NDIAG;
	NodeErr4_K:= 	MODULES03[4].CH_NDIAG;
	NodeErr5_K:= 	MODULES03[5].CH_NDIAG;
	NodeErr6_K:= 	MODULES03[6].CH_NDIAG;
	NodeErr7_K:= 	MODULES03[7].CH_NDIAG;
	NodeErr8_K:= 	MODULES03[8].CH_NDIAG;
	NodeErr9_K:= 	MODULES03[9].CH_NDIAG;
	NodeErr10_K:= 	MODULES03[10].CH_NDIAG;
	NodeErr11_K:= 	MODULES03[11].CH_NDIAG;
	NodeErr12_K:= 	MODULES03[12].CH_NDIAG;
	NodeErr13_K:= 	MODULES03[13].CH_NDIAG;
	NodeErr14_K:= 	MODULES03[14].CH_NDIAG;
	NodeErr15_K:= 	MODULES03[15].CH_NDIAG;
	NodeErr16_K:= 	MODULES03[16].CH_NDIAG;

	CfgErr1_K:=	 	MODULES03[1].CH_MODCONF;
	CfgErr2_K:=	 	MODULES03[2].CH_MODCONF;
	CfgErr3_K:=	 	MODULES03[3].CH_MODCONF;
	CfgErr4_K:=	 	MODULES03[4].CH_MODCONF;
	CfgErr5_K:=	 	MODULES03[5].CH_MODCONF;
	CfgErr6_K:=	 	MODULES03[6].CH_MODCONF;
	CfgErr7_K:=	 	MODULES03[7].CH_MODCONF;
	CfgErr8_K:=	 	MODULES03[8].CH_MODCONF;
	CfgErr9_K:=	 	MODULES03[9].CH_MODCONF;
	CfgErr10_K:=	MODULES03[10].CH_MODCONF;
	CfgErr11_K:=	MODULES03[11].CH_MODCONF;
	CfgErr12_K:=	MODULES03[12].CH_MODCONF;
	CfgErr13_K:=	MODULES03[13].CH_MODCONF;
	CfgErr14_K:=	MODULES03[14].CH_MODCONF;
	CfgErr15_K:=	MODULES03[15].CH_MODCONF;
	CfgErr16_K:=	MODULES03[16].CH_MODCONF;

END_PROGRAM

// REZERV1/REZERV1
PROGRAM REZERV1
VAR CONSTANT
	Timeout_NoPila_FromNet:TIME:=T#1500MS;//T#2000MS;
	Timeout_NoPila_FromCOM:TIME:=T#1500MS;//T#2000MS;
	Timeout_NoPila_FromNetBoth:TIME:=T#500MS;//
	Timeout_NoPila_FromCOMBoth:TIME:=T#500MS;//
	Imp_U24:TIME:=T#1000MS;//импульс включения реле U+24
	ImpLong_U24:TIME:=T#3000MS;//импульс подавления паразитного переключения реле U+24 при включении другого контроллера
	// макс значение счетчика тактов задачи, через которые повторяется импульс на реле +24В от Active/Single
	Redire_Udo_CntMax:WORD:=300;// макс значение (100 = 10сек) (300 = 30сек)
END_VAR
VAR
	// для работы кнопок из визуализации
	StopMyPila:BOOL;// =1 - остановить мою пилу
	StopMyPilaStatus:BOOL;// =1 - остановить мою пилу Статуса
	StopMyPilaReady:BOOL;// =1 - остановить мою пилу Готовности
	//
	StopMyPilaAktiv:BOOL;// =1 - остановить мою пилу Активности для формирования меандра акт на DO
	//

	BMPERR1:WORD;// ошибки УСО этого контроллера

	Tst1:PilaTst;// функц-блок наличия пилы соседа (сеть)
	Tst2:PilaTst;// функц-блок наличия пилы соседа (COM)
	Tst1Both:PilaTst;// функц-блок наличия пилы соседа (сеть)- для фиксации отсутствия пил по обоим каналам
	Tst2Both:PilaTst;// функц-блок наличия пилы соседа (COM)- для фиксации отсутствия пил по обоим каналам
	
	StateK:RezervState;// Статус контроллера
	ReadyK:WORD;// Готовность к управлению
	Cmd_GoPassive:WORD;// команда "Стать пассивным" (от МПУ или из-вне)

	My_Udo:BOOL:=FALSE;// Вкл/откл U пит +24В на DO - внутреннее использование для формирования импульса
	Udo:BOOL:=FALSE;// Вкл/откл U пит +24В на DO
	MasterOPC:BOOL:=FALSE;// Мастер-переменная ОРС

	StateStr:STRING;
	ReadyStr:WSTRING;
	
	My_MX_Mode:WORD;// выходная переменная как MX_Mode
	My_MX_Status:WORD;// входная переменная как MX_Status

	// управление переключением каналов резервирования: сеть/COM
	NoPila_FromNet:BOOL;// признак отсутствия пилы соседа по сети
	NoPila_FromCOM:BOOL;// признак отсутствия пилы соседа по COM
	NoPila_FromREZ:BOOL;// признак отсутствия пилы соседа из подпрограммы REZ1 или REZ2 (суммарно по трем пилам, по NET, по COM) 
	NoPila_FromNetBoth:BOOL;// признак отсутствия пилы соседа по сети (для одновременного отсут обоих пил)
	NoPila_FromCOMBoth:BOOL;// признак отсутствия пилы соседа по COM (для одновременного отсут обоих пил)
	

	REZZ1:REZ1;
	WDOG_Go:WORD;
	WDOG_T:TON;
	
	TP_Udo:TP;// формирование импульса на переключение реле U+24
	TP2_Udo:TP;// формирование импульса на переключение реле U+24 при старте другого контроллера
	
	Index_PROG1:INT:=0;
	StateK_BlinkCnt:INT:=0;
	
	Redire_Udo_Cnt:WORD:=1;// счетчик тактов задачи, через которые повторяется импульс на реле +24В от Active/Single
	
	PilaAktiv:WORD;// счетчик для формирования меандра активности физического выхода DO
END_VAR

///////////////////////////////////////////////////////////////////////////////////////////////////
// включить использование моей версии СОМ-порта
//{define Use_MyCOM_in_Rezerv}
// отключить использование моей версии СОМ-порта
{undefine Use_MyCOM_in_Rezerv}

// выдать в окно "Message" подсказку
{IF defined (Use_MyCOM_in_Rezerv) }
{info 'Use my COM-rezerv in program'}
{ELSE}
{info 'Use COM-rezerv in RWH driver'}
{END_IF}
///////////////////////////////////////////////////////////////////////////////////////////////////

///////////////////////////////////////////////////////////////////////////////////////////////////
// включить использование импульса для переключения реле питания +24В
{define Use_U24Imp_in_Rezerv}
// отключить использование импульса для переключения реле питания +24В
//{undefine Use_U24Imp_in_Rezerv}

// выдать в окно "Message" подсказку
{IF defined (Use_U24Imp_in_Rezerv) }
{info 'Use Imp for Udo=+24'}
{ELSE}
{info 'NOT Use Imp for Udo=+24'}
{END_IF}
///////////////////////////////////////////////////////////////////////////////////////////////////

///////////////////////////////////////////////////////////////////////////////////////////////////
// включить импульс для подавления паразитного переключения реле питания +24В при включении другого контроллера
{define Use_U24ImpOnStart_in_Rezerv}
// отключить импульс для подавления паразитного переключения реле питания +24В при включении другого контроллера
//{undefine Use_U24ImpOnStart_in_Rezerv}
// импульс выдается по включению блока питания соседнего контоллера

// выдать в окно "Message" подсказку
{IF defined (Use_U24ImpOnStart_in_Rezerv) }
{info 'Use Imp for Udo=+24 on Start Controller'}
{ELSE}
{info 'NOT Use Imp for Udo=+24 on Start Controller'}
{END_IF}
///////////////////////////////////////////////////////////////////////////////////////////////////

///////////////////////////////////////////////////////////////////////////////////////////////////
// включить использование импульса для переключения реле питания +24В во всех режимах,кроме Single
{define Use_U24ImpNotOnlySingleMode_in_Rezerv}
// отключить использование импульса для переключения реле питания +24В во всех режимах,кроме Single
//{undefine Use_U24ImpNotOnlySingleMode_in_Rezerv}
// в режиме Single использовать потенциальный сигнал, а в режимах Active, Passive - импульс

// выдать в окно "Message" подсказку
{IF defined (Use_U24ImpNotOnlySingleMode_in_Rezerv) }
{info 'Use Imp for Udo=+24 only Active and Passive Mode'}
{ELSE}
{info 'NOT Use Imp for Udo=+24 only Active and Passive Mode'}
{END_IF}
///////////////////////////////////////////////////////////////////////////////////////////////////

///////////////////////////////////////////////////////////////////////////////////////////////////
// включить периодический импульс подтверждения установки реле питания +24В в режимах Active/Single
{define Use_U24ImpRedire_in_Rezerv}
// отключить периодический импульс подтверждения установки реле питания +24В в режимах Active/Single
//{undefine Use_U24ImpRedire_in_Rezerv}
// импульс выдается каждые Redire_Udo_CntMax циклов задачи

// выдать в окно "Message" подсказку
{IF defined (Use_U24ImpRedire_in_Rezerv) }
{info 'Use Imp Redire for Udo=+24'}
{ELSE}
{info 'NOT Use Imp Redire for Udo=+24'}
{END_IF}
///////////////////////////////////////////////////////////////////////////////////////////////////

CASE Index_PROG1 OF
0:// инициализация
	Index_PROG1:=1;

1:
(*
// Это для рестарта контроллера из инстр системы - поставить 16#55AC и отключить сразу (LOGOUT) 
IF WDOG_Go=16#55AC
	THEN
	WDOG_T(In:=1, PT:=TIME#5S);
	IF WDOG_T.Q
		THEN
		%QW13:=WDOG_Go;		//		MainUP_PRG.WDOG_O:=WDOG_Go;
	END_IF
END_IF
*)


// формировать пилу жизни
IF NOT StopMyPila
	THEN
	IF PilaK1_O < 100
		THEN
		PilaK1_O:=PilaK1_O+1;
		ELSE
		PilaK1_O:=0;		
	END_IF
END_IF



IF NOT StopMyPilaStatus
	THEN
	StatusK1_O:= (PilaK1_O AND 16#FF)+ (StateK*256);// выдать свой статус в сеть в старшем байте и пилу в младшем байте
END_IF



IF NOT StopMyPilaReady
	THEN
	ReadyK1_O:= (PilaK1_O AND 16#FF)+ (ReadyK*256);// выдать свою готовность в сеть в старшем байте и пилу в младшем байте
END_IF

{IF defined (Use_MyCOM_in_Rezerv) }
{ELSE}
	// выдать в COM-rezerv in RWH-driver			
	%QW16:=PilaK1_O;
	%QW17:=StatusK1_O;
	%QW18:=ReadyK1_O;
{END_IF}

///////////////////////////////////////////////////////////////////////////////////////////////////
// Контроль пил для фиксации отключения контроллера - нет пилы Net и нет пилы COM одновременно
	Tst1Both(Pila:=PilaK2_O, TimeOut:=Timeout_NoPila_FromNetBoth, NoPila=>NoPila_FromNetBoth);
{IF defined (Use_MyCOM_in_Rezerv) }
		// для использования с моим COM-портом !!!
	Tst2Both(Pila:=COM102_PRG.PilaFromK2, TimeOut:=Timeout_NoPila_FromCOMBoth, NoPila=>NoPila_FromCOMBoth);
{ELSE}
	Tst2Both(Pila:=%IW16, TimeOut:=Timeout_NoPila_FromCOMBoth, NoPila=>NoPila_FromCOMBoth);
{END_IF}
///////////////////////////////////////////////////////////////////////////////////////////////////


///////////////////////////////////////////////////////////////////////////////////////////////////
// Контроль пил для переключения каналов резервирования: Net - COM
	Tst1(Pila:=PilaK2_O, TimeOut:=Timeout_NoPila_FromNet, NoPila=>NoPila_FromNet);
{IF defined (Use_MyCOM_in_Rezerv) }
		// для использования с моим COM-портом !!!
	Tst2(Pila:=COM102_PRG.PilaFromK2, TimeOut:=Timeout_NoPila_FromCOM, NoPila=>NoPila_FromCOM);
{ELSE}
	Tst2(Pila:=%IW16, TimeOut:=Timeout_NoPila_FromCOM, NoPila=>NoPila_FromCOM);
{END_IF}
///////////////////////////////////////////////////////////////////////////////////////////////////

	
	IF NOT NoPila_FromNet
		THEN//есть пила по NET - работаем по сети
		REZZ1(_BMPERR:={BMPERR1}BMPERR_I, _My_MX_Status:={My_MX_Status}MxStatus_I, 
				_PilaK_O:= PilaK2_O, _StatusK_O:=StatusK2_O, _ReadyK_O:=ReadyK2_O,
				 _NumK:=1,// это контроллер №1
					_StateK:=StateK, _ReadyK:=ReadyK, _Cmd_GoPassive:=Cmd_GoPassive,
					_NoPilaBoth:=NoPila_FromCOMBoth AND NoPila_FromNetBoth AND (MxStatus_I.15),// 02 ноя 2012
					_NoPilaCommon=>NoPila_FromREZ, 
					_My_MX_Mode=>{My_MX_Mode}{%QW1}MxMode_O, _Udo=>My_Udo, _MasterOPC=>MasterOPC, _StateStr=>StateStr, _ReadyStr=>ReadyStr);
		
		ELSE//нет пилы по NET - работаем по СОМ
{IF defined (Use_MyCOM_in_Rezerv) }
		// для использования с моим COM-портом !!!
		// 	сделать задачи TaskCOM (запускает COM102_PRG), TaskCOM101(запускает COM101_PRG) в К1
		//     и задачи TaskCOM(запускает COM202_PRG), TaskCOM201(запускает COM201_PRG) в К2
		REZZ1(_BMPERR:={BMPERR1}BMPERR_I, _My_MX_Status:={My_MX_Status}MxStatus_I,
				_PilaK_O:= COM102_PRG.PilaFromK2, _StatusK_O:= COM102_PRG.StatusFromK2, _ReadyK_O:= COM102_PRG.ReadyFromK2,
				 _NumK:=1,// это контроллер №1
					_StateK:=StateK, _ReadyK:=ReadyK, _Cmd_GoPassive:=Cmd_GoPassive,
					_NoPilaBoth:=NoPila_FromCOMBoth AND NoPila_FromNetBoth AND (MxStatus_I.15),// 02 ноя 2012
					_NoPilaCommon=>NoPila_FromREZ, 
					_My_MX_Mode=>{My_MX_Mode}{%QW1}MxMode_O, _Udo=>My_Udo, _MasterOPC=>MasterOPC, _StateStr=>StateStr, _ReadyStr=>ReadyStr);
{ELSE}
		REZZ1(_BMPERR:={BMPERR1}BMPERR_I, _My_MX_Status:={My_MX_Status}MxStatus_I,
				_PilaK_O:= %IW16, _StatusK_O:= %IW17, _ReadyK_O:= %IW18,
				 _NumK:=1,// это контроллер №1
					_StateK:=StateK, _ReadyK:=ReadyK, _Cmd_GoPassive:=Cmd_GoPassive,
					_NoPilaBoth:=NoPila_FromCOMBoth AND NoPila_FromNetBoth AND (MxStatus_I.15),// 02 ноя 2012
					_NoPilaCommon=>NoPila_FromREZ,					
					_My_MX_Mode=>{My_MX_Mode}{%QW1}MxMode_O, _Udo=>My_Udo, _MasterOPC=>MasterOPC, _StateStr=>StateStr, _ReadyStr=>ReadyStr);
{END_IF}
	END_IF


//////// добавлено вместо закомментированого 8 апр 2013//////исправляем включение другого К ///////////////////////////
{IF defined (Use_U24Imp_in_Rezerv) }
// импульсное управление Udo	

	{IF defined (Use_U24ImpNotOnlySingleMode_in_Rezerv) }
	// импульсное управление Udo в режимах Active и Passive, но потенциальное удержание в Single	
		IF (StateK=Active)OR(StateK=Passive)
			THEN
			TP_Udo(in:=My_Udo, pt:=Imp_U24, Q=>Udo);
		END_IF
		IF (StateK=Single)
			THEN
			Udo:=My_Udo;	
		END_IF
	{ELSE}
			TP_Udo(in:=My_Udo, pt:=Imp_U24, Q=>Udo);
	{END_IF}

	{IF defined (Use_U24ImpRedire_in_Rezerv) }	
	// Периодический импульс подтверждения установки реле питания +24В в режимах Active/Single (добавлено 9 апр 2013)
	IF (StateK=Active)OR(StateK=Single)
		THEN
		IF (Redire_Udo_Cnt < Redire_Udo_CntMax)
			THEN
				Redire_Udo_Cnt:=Redire_Udo_Cnt+1;
			ELSE
				Redire_Udo_Cnt:=0;
				Udo:=1;
		END_IF
	END_IF
	{END_IF}
	
	{IF defined (Use_U24ImpOnStart_in_Rezerv)}
	// Импульс для подавления паразитного переключения Udo при включении другого контроллера
	IF (StateK=Active)OR(StateK=Single)
		THEN
		TP2_Udo(in:=DI_K[{11}9].RR.1, pt:=ImpLong_U24);
		IF TP2_Udo.Q
			THEN
			Udo:=1;
		END_IF
	END_IF
	{END_IF}
	
{ELSE}
// без импульса - потенциальное управление Udo	
	Udo:=My_Udo;	
{END_IF}
//////// окончание добавленого вместо закомментированого 8 апр 2013//////исправляем включение другого К ///////////////

	// в Помарской не прописан Udo прямо во вкладке DO поз.4 (как в ГавЯм DO_bit3 поз.16) - Фалеев 29.05.2018
	DO_K[3].RR.3:=	Udo;// подать напр на выходы	

	// в Помарской пилу активности для меандра
	//StopMyPilaAktiv  :=	NOT ((StateK=Single)OR(StateK=Active));// остановить пилу только в пассиве		- закоммент. 31 мая 2018 Фалеев
	StopMyPilaAktiv  :=	((StateK=Active)AND((ReadyK2_O AND 16#FF00)=0)AND(BMPERR_I.7)) OR	// Я активный, другой (K2) не готов и у меня есть ошибка АВ УСО (поз8) - остановить пилу АКТ.
						((StateK=Single)AND (BMPERR_I.7)) OR				// Я один и у меня есть ошибка АВ УСО (поз8) - остановить пилу АКТ.
						(StateK=Passive)OR(StateK=Nothing);					// Я пассивный или ничего - остановить пилу АКТ.
	
	// формировать пилу активности для меандра акт DO
	IF NOT StopMyPilaAktiv
		THEN
			PilaAktiv:=PilaAktiv+1;
	END_IF
	DO_K[3].RR.0:=	PilaAktiv.0;	// вывести в DO3_bit0	 меандр активности   поз.4
	DO_K[3].RR.11:=	PilaAktiv.0;	// вывести в DO3_bit11	 (для К1 индикация на дверь)   поз.4
	//DO_K[3].RR.12:=	PilaAktiv.0;	// вывести в DO3_bit12	 (для К2 индикация на дверь)   поз.4


// просто индикация для   ПОМАРСКОЙ   !!!   поз.2
	DO_K[2].RR.8:=NoPila_FromNet;
	DO_K[2].RR.9:=NoPila_FromCOM;
	DO_K[2].RR.11:=Udo;// подать напр на выходы	
	DO_K[2].RR.13:=(BMPERR_I <> 0);
	DO_K[2].RR.15:=NoPila_FromREZ;

	CASE StateK OF
 	Single:
			DO_K[2].RR.10:= 1;// Single
			DO_K[2].RR.12:= 0;// Active
			DO_K[2].RR.14:= 0;// Passive

	Active:	
			DO_K[2].RR.10:= 0;// Single
			DO_K[2].RR.12:= 1;// Active
			DO_K[2].RR.14:= 0;// Passive
	
	Passive:
			DO_K[2].RR.10:= 0;// Single
			DO_K[2].RR.12:= 0;// Active
			DO_K[2].RR.14:= 1;// Passive
	
	END_CASE	

	
END_CASE

END_PROGRAM

// K2/std12k5/Elpk_03_02/MainUP_PRG
PROGRAM MainUP_PRG
VAR
	START_INDEX, INDEX, INDEX2:INT:=0;
	
	I1,I2,I3,I4,I5,I6:INT;
	J1,J2,J3,J4,J5,J6,J7,J8,J9:INT;
	WWW1, WWW2, WWW3, WWW4, WWW5, WWW6, WWW7, WWW8:WORD;
	//ERR1, ERR2, ERR3, ERR4, ERR5, ERR6, ERR7, ERR8, ERR9, ERR22:RTS_IEC_RESULT;
	//ERR101, ERR102, ERR103, ERR104, ERR105,  ERR122:RTS_IEC_RESULT;
	//szFile1,szFile2:REFERENCE TO STRING;
	WW_WW1, WW_WW2, WW_WW3, WW_WW4:WORD;
	

//	GEN1:GEN;
//	IGEN1:INT;
/////////////////////////////////////////////////////////////////////////////////////////////////////////////
   {attribute 'displaymode':='hex'}
	MxStatus:WORD;		// OPC
//   {attribute 'displaymode':='hex'}
//	MxStatus_I:WORD;		// внутреннее использование

   {attribute 'displaymode':='hex'}
	MxMode:WORD;		// MX Active = 8
   {attribute 'displaymode':='hex'}
	//MxMode_O:WORD;		// внутреннее использование

	ADCWAY_I:WORD;
	ADCWAY_II:WORD;		// внутреннее использование
	
	ADCWAY_O:WORD;
	ADCWAY_OO:WORD;		// внутреннее использование

   {attribute 'displaymode':='hex'}
	BMPPRES:WORD;		// OPC
//   {attribute 'displaymode':='hex'}
//	BMPPRES_I:WORD;		// внутреннее использование

   {attribute 'displaymode':='hex'}
	BMPERR:WORD;		// OPC
///   {attribute 'displaymode':='hex'}
///	BMPERR_I:WORD;		// внутреннее использование

	MXLINES_I:WORD;
	MXLINES:WORD;
	
	HIDE_ERR_OUT_I:WORD;
	HIDE_ERR_OUT_II:WORD;

	HIDE_ERR_OUT_O:WORD;
	HIDE_ERR_OUT_OO:WORD;
	RWH_PERIOD_I:WORD;
	RWH_PERIOD:WORD;

	MX_ATT_I:WORD;
	MX_ATT:WORD;

	EXTCMD_I:WORD;
	EXTCMD:WORD;
   {attribute 'displaymode':='hex'}
	WDOG_O:WORD;
	
	
	
	
	// для отладки
   {attribute 'displaymode':='hex'}
	CH_MODCONF:WORD;
   {attribute 'displaymode':='hex'}
	CH_ERRNOW:WORD;
   {attribute 'displaymode':='hex'}
	CH_ERRHIST:WORD;
   {attribute 'displaymode':='hex'}
	CH_NDIAG:WORD;
   {attribute 'displaymode':='hex'}
	CH_MDIAG:WORD;
   {attribute 'displaymode':='hex'}
	CH_FIRMVER:WORD;
   {attribute 'displaymode':='hex'}
	CH_FIRMDATE:WORD;
   {attribute 'displaymode':='hex'}
	CH_CH7:WORD;
	// конец для отладки
(*
	MODULE_01:T_DIAGNOSTIC;
	MODULE_02:T_DIAGNOSTIC;
	MODULE_03:T_DIAGNOSTIC;
	MODULE_04:T_DIAGNOSTIC;
	MODULE_05:T_DIAGNOSTIC;
	MODULE_06:T_DIAGNOSTIC;
	MODULE_07:T_DIAGNOSTIC;
	MODULE_08:T_DIAGNOSTIC;
	MODULE_09:T_DIAGNOSTIC;
	MODULE_10:T_DIAGNOSTIC;
	MODULE_11:T_DIAGNOSTIC;
	MODULE_12:T_DIAGNOSTIC;
	MODULE_13:T_DIAGNOSTIC;
	MODULE_14:T_DIAGNOSTIC;
	MODULE_15:T_DIAGNOSTIC;
	MODULE_16:T_DIAGNOSTIC;
	*)

(*
   {attribute 'displaymode':='hex'}
	NodeErr1:WORD;	// OPC		
	///NodeErr1_Log:AddLOG_W_UP;// FB для записи NodeErr в лог при изменении значения	
   {attribute 'displaymode':='hex'}
	NodeErr2:WORD;	// OPC	
	///NodeErr2_Log:AddLOG_W_UP;// FB для записи NodeErr в лог при изменении значения	
   {attribute 'displaymode':='hex'}
	NodeErr3:WORD;	// OPC	
	///NodeErr3_Log:AddLOG_W_UP;// FB для записи NodeErr в лог при изменении значения	
   {attribute 'displaymode':='hex'}
	NodeErr4:WORD;	// OPC	
	///NodeErr4_Log:AddLOG_W_UP;// FB для записи NodeErr в лог при изменении значения	
   {attribute 'displaymode':='hex'}
	NodeErr5:WORD;	// OPC	
	///NodeErr5_Log:AddLOG_W_UP;// FB для записи NodeErr в лог при изменении значения	
   {attribute 'displaymode':='hex'}
	NodeErr6:WORD;	// OPC	
	///NodeErr6_Log:AddLOG_W_UP;// FB для записи NodeErr в лог при изменении значения	
   {attribute 'displaymode':='hex'}
	NodeErr7:WORD;	// OPC	
	///NodeErr7_Log:AddLOG_W_UP;// FB для записи NodeErr в лог при изменении значения	
   {attribute 'displaymode':='hex'}
	NodeErr8:WORD;	// OPC	
	///NodeErr8_Log:AddLOG_W_UP;// FB для записи NodeErr в лог при изменении значения	
   {attribute 'displaymode':='hex'}
	NodeErr9:WORD;	// OPC	
	///NodeErr9_Log:AddLOG_W_UP;// FB для записи NodeErr в лог при изменении значения	
   {attribute 'displaymode':='hex'}
	NodeErr10:WORD;	// OPC
	///NodeErr10_Log:AddLOG_W_UP;// FB для записи NodeErr в лог при изменении значения	
   {attribute 'displaymode':='hex'}
	NodeErr11:WORD;	// OPC
	///NodeErr11_Log:AddLOG_W_UP;// FB для записи NodeErr в лог при изменении значения	
   {attribute 'displaymode':='hex'}
	NodeErr12:WORD;	// OPC
	///NodeErr12_Log:AddLOG_W_UP;// FB для записи NodeErr в лог при изменении значения	
   {attribute 'displaymode':='hex'}
	NodeErr13:WORD;	// OPC
	///NodeErr13_Log:AddLOG_W_UP;// FB для записи NodeErr в лог при изменении значения	
   {attribute 'displaymode':='hex'}
	NodeErr14:WORD;	// OPC
	///NodeErr14_Log:AddLOG_W_UP;// FB для записи NodeErr в лог при изменении значения	
   {attribute 'displaymode':='hex'}
	NodeErr15:WORD;	// OPC
	///NodeErr15_Log:AddLOG_W_UP;// FB для записи NodeErr в лог при изменении значения	
   {attribute 'displaymode':='hex'}
	NodeErr16:WORD;	// OPC
	///NodeErr16_Log:AddLOG_W_UP;// FB для записи NodeErr в лог при изменении значения	

	///ImitatorON_Log:AddLOG_W_UP;// FB для записи в лог при изменении значения	

*)
END_VAR

// только для тестирования !!!
(*od.do_1.bits[0]:=0;*)
(*od.do_1.bits[1]:=1;
od.do_1.bits[2]:=1;
od.do_1.bits[3]:=1;
od.do_1.bits[4]:=1;
od.do_1.bits[5]:=1;
od.do_1.bits[6]:=1;
od.do_1.bits[7]:=1;

od.do_1.bits[8]:=1;
od.do_1.bits[9]:=1;
od.do_1.bits[10]:=1;
od.do_1.bits[11]:=1;
od.do_1.bits[12]:=1;
od.do_1.bits[13]:=1;
od.do_1.bits[14]:=1;
od.do_1.bits[15]:=1;
*)






	//
	// Формирование пилы жизни для передачи в ОРС. Значения от 0 до 1023. На каждом цикле +1.
	//
	LifeCnt:= (LifeCnt+1)AND 16#3FF;


///////////////////////////////////////////////////////////////////////////////////////////////////
//	Читать диагностику

	MxStatus:=MxStatus_I;	// OPC

	ADCWAY_II:=ADCWAY_I;
	BMPPRES_K:= BMPPRES:= BMPPRES_I;// в ОРС


	(*IF Imitator_code=16#55AA
	THEN// если есть имитатор - брать диагностику из имитатора и передать а ОРС
		BMPERR:=BMPERR_UP1_Im;// в ОРС
	ELSE
	// нет имитатора - брать диагностику из драйвера и передать в ОРС
		BMPERR:=BMPERR_I;// в ОРС
	END_IF
	BMPERR_K:=	BMPERR;*)
	BMPERR_K:=	BMPERR:=	BMPERR_I;// в ОРС

		
	MXLINES:=MXLINES_I;
	HIDE_ERR_OUT_II:=HIDE_ERR_OUT_I;
	RWH_PERIOD:=RWH_PERIOD_I;
	MX_ATT:=MX_ATT_I;
	EXTCMD:=EXTCMD_I;
	
//	ADCWAY_O:=%QW2;
//	HIDE_ERR_OUT_O:=%QW9;
//	WDOG_O:=16#55AA;	// Включить watchdog



	MasterOPC_ST:=REZERV2.MasterOPC;
	
	
	NodeErr1_K:= 	MODULES03[1].CH_NDIAG;
	NodeErr2_K:= 	MODULES03[2].CH_NDIAG;
	NodeErr3_K:= 	MODULES03[3].CH_NDIAG;
	NodeErr4_K:= 	MODULES03[4].CH_NDIAG;
	NodeErr5_K:= 	MODULES03[5].CH_NDIAG;
	NodeErr6_K:= 	MODULES03[6].CH_NDIAG;
	NodeErr7_K:= 	MODULES03[7].CH_NDIAG;
	NodeErr8_K:= 	MODULES03[8].CH_NDIAG;
	NodeErr9_K:= 	MODULES03[9].CH_NDIAG;
	NodeErr10_K:= 	MODULES03[10].CH_NDIAG;
	NodeErr11_K:= 	MODULES03[11].CH_NDIAG;
	NodeErr12_K:= 	MODULES03[12].CH_NDIAG;
	NodeErr13_K:= 	MODULES03[13].CH_NDIAG;
	NodeErr14_K:= 	MODULES03[14].CH_NDIAG;
	NodeErr15_K:= 	MODULES03[15].CH_NDIAG;
	NodeErr16_K:= 	MODULES03[16].CH_NDIAG;

	CfgErr1_K:=	 	MODULES03[1].CH_MODCONF;
	CfgErr2_K:=	 	MODULES03[2].CH_MODCONF;
	CfgErr3_K:=	 	MODULES03[3].CH_MODCONF;
	CfgErr4_K:=	 	MODULES03[4].CH_MODCONF;
	CfgErr5_K:=	 	MODULES03[5].CH_MODCONF;
	CfgErr6_K:=	 	MODULES03[6].CH_MODCONF;
	CfgErr7_K:=	 	MODULES03[7].CH_MODCONF;
	CfgErr8_K:=	 	MODULES03[8].CH_MODCONF;
	CfgErr9_K:=	 	MODULES03[9].CH_MODCONF;
	CfgErr10_K:=	MODULES03[10].CH_MODCONF;
	CfgErr11_K:=	MODULES03[11].CH_MODCONF;
	CfgErr12_K:=	MODULES03[12].CH_MODCONF;
	CfgErr13_K:=	MODULES03[13].CH_MODCONF;
	CfgErr14_K:=	MODULES03[14].CH_MODCONF;
	CfgErr15_K:=	MODULES03[15].CH_MODCONF;
	CfgErr16_K:=	MODULES03[16].CH_MODCONF;

END_PROGRAM

// REZERV1/REZERV2
PROGRAM REZERV2
VAR CONSTANT
	Timeout_NoPila_FromNet:TIME:=T#1500MS;//T#2000MS;
	Timeout_NoPila_FromCOM:TIME:=T#1500MS;//T#2000MS;
	Timeout_NoPila_FromNetBoth:TIME:=T#500MS;//
	Timeout_NoPila_FromCOMBoth:TIME:=T#500MS;//
	Imp_U24:TIME:=T#1000MS;//импульс включения реле U+24
	ImpLong_U24:TIME:=T#3000MS;//импульс подавления паразитного переключения реле U+24 при включении другого контроллера
	// макс значение счетчика тактов задачи, через которые повторяется импульс на реле +24В от Active/Single
	Redire_Udo_CntMax:WORD:=300;// макс значение (100 = 10сек) (300 = 30сек)
END_VAR
VAR
	// для работы кнопок из визуализации
	StopMyPila:BOOL;// =1 - остановить мою пилу
	StopMyPilaStatus:BOOL;// =1 - остановить мою пилу Статуса
	StopMyPilaReady:BOOL;// =1 - остановить мою пилу Готовности
	//
	StopMyPilaAktiv:BOOL;// =1 - остановить мою пилу Активности для формирования меандра акт на DO
	//

	BMPERR2:WORD;// ошибки УСО этого контроллера

	Tst1:PilaTst;// функц-блок наличия пилы соседа (сеть)
	Tst2:PilaTst;// функц-блок наличия пилы соседа (COM)
	Tst1Both:PilaTst;// функц-блок наличия пилы соседа (сеть)- для фиксации отсутствия пил по обоим каналам
	Tst2Both:PilaTst;// функц-блок наличия пилы соседа (COM)- для фиксации отсутствия пил по обоим каналам
	
	StateK:RezervState;// Статус контроллера
	ReadyK:WORD;// Готовность к управлению
	Cmd_GoPassive:WORD;// команда "Стать пассивным" (от МПУ или из-вне)

	My_Udo:BOOL:=FALSE;// Вкл/откл U пит +24В на DO - внутреннее использование для формирования импульса
	Udo:BOOL:=FALSE;// Вкл/откл U пит +24В на DO
	MasterOPC:BOOL:=FALSE;// Мастер-переменная ОРС

	StateStr:STRING;
	ReadyStr:WSTRING;
	
	My_MX_Mode:WORD;// выходная переменная как MX_Mode
	My_MX_Status:WORD;// входная переменная как MX_Status

	// управление переключением каналов резервирования: сеть/COM
	NoPila_FromNet:BOOL;// признак отсутствия пилы соседа по сети
	NoPila_FromCOM:BOOL;// признак отсутствия пилы соседа по COM
	NoPila_FromREZ:BOOL;// признак отсутствия пилы соседа из подпрограммы REZ1 или REZ2 (суммарно по трем пилам, по NET, по COM) 
	NoPila_FromNetBoth:BOOL;// признак отсутствия пилы соседа по сети (для одновременного отсут обоих пил)
	NoPila_FromCOMBoth:BOOL;// признак отсутствия пилы соседа по COM (для одновременного отсут обоих пил)
	

	REZZ1:REZ1;
	WDOG_Go:WORD;
	WDOG_T:TON;
	
	TP_Udo:TP;// формирование импульса на переключение реле U+24
	TP2_Udo:TP;// формирование импульса на переключение реле U+24 при старте другого контроллера
	
	Index_PROG2:INT:=0;
	StateK_BlinkCnt:INT:=0;
	
	Redire_Udo_Cnt:WORD:=1;// счетчик тактов задачи, через которые повторяется импульс на реле +24В от Active/Single
	
	PilaAktiv:WORD;// счетчик для формирования меандра активности физического выхода DO
END_VAR

///////////////////////////////////////////////////////////////////////////////////////////////////
// включить использование моей версии СОМ-порта
//{define Use_MyCOM_in_Rezerv}
// отключить использование моей версии СОМ-порта
{undefine Use_MyCOM_in_Rezerv}

// выдать в окно "Message" подсказку
{IF defined (Use_MyCOM_in_Rezerv) }
{info 'Use my COM-rezerv in program'}
{ELSE}
{info 'Use COM-rezerv in RWH driver'}
{END_IF}
///////////////////////////////////////////////////////////////////////////////////////////////////

///////////////////////////////////////////////////////////////////////////////////////////////////
// включить использование импульса для переключения реле питания +24В
{define Use_U24Imp_in_Rezerv}
// отключить использование импульса для переключения реле питания +24В
//{undefine Use_U24Imp_in_Rezerv}

// выдать в окно "Message" подсказку
{IF defined (Use_U24Imp_in_Rezerv) }
{info 'Use Imp for Udo=+24'}
{ELSE}
{info 'NOT Use Imp for Udo=+24'}
{END_IF}
///////////////////////////////////////////////////////////////////////////////////////////////////

///////////////////////////////////////////////////////////////////////////////////////////////////
// включить импульс для подавления паразитного переключения реле питания +24В при включении другого контроллера
{define Use_U24ImpOnStart_in_Rezerv}
// отключить импульс для подавления паразитного переключения реле питания +24В при включении другого контроллера
//{undefine Use_U24ImpOnStart_in_Rezerv}
// импульс выдается по включению блока питания соседнего контоллера

// выдать в окно "Message" подсказку
{IF defined (Use_U24ImpOnStart_in_Rezerv) }
{info 'Use Imp for Udo=+24 on Start Controller'}
{ELSE}
{info 'NOT Use Imp for Udo=+24 on Start Controller'}
{END_IF}
///////////////////////////////////////////////////////////////////////////////////////////////////

///////////////////////////////////////////////////////////////////////////////////////////////////
// включить использование импульса для переключения реле питания +24В во всех режимах,кроме Single
{define Use_U24ImpNotOnlySingleMode_in_Rezerv}
// отключить использование импульса для переключения реле питания +24В во всех режимах,кроме Single
//{undefine Use_U24ImpNotOnlySingleMode_in_Rezerv}
// в режиме Single использовать потенциальный сигнал, а в режимах Active, Passive - импульс

// выдать в окно "Message" подсказку
{IF defined (Use_U24ImpNotOnlySingleMode_in_Rezerv) }
{info 'Use Imp for Udo=+24 only Active and Passive Mode'}
{ELSE}
{info 'NOT Use Imp for Udo=+24 only Active and Passive Mode'}
{END_IF}
///////////////////////////////////////////////////////////////////////////////////////////////////

///////////////////////////////////////////////////////////////////////////////////////////////////
// включить периодический импульс подтверждения установки реле питания +24В в режимах Active/Single
{define Use_U24ImpRedire_in_Rezerv}
// отключить периодический импульс подтверждения установки реле питания +24В в режимах Active/Single
//{undefine Use_U24ImpRedire_in_Rezerv}
// импульс выдается каждые Redire_Udo_CntMax циклов задачи

// выдать в окно "Message" подсказку
{IF defined (Use_U24ImpRedire_in_Rezerv) }
{info 'Use Imp Redire for Udo=+24'}
{ELSE}
{info 'NOT Use Imp Redire for Udo=+24'}
{END_IF}
///////////////////////////////////////////////////////////////////////////////////////////////////

CASE Index_PROG2 OF
0:// инициализация
	Index_PROG2:=1;

1:
(*
// Это для рестарта контроллера из инстр системы - поставить 16#55AC и отключить сразу (LOGOUT) 
IF WDOG_Go=16#55AC
	THEN
	WDOG_T(In:=1, PT:=TIME#5S);
	IF WDOG_T.Q
		THEN
		%QW13:=WDOG_Go;
	END_IF
END_IF
*)


// формировать пилу жизни
IF NOT StopMyPila
	THEN
	IF PilaK2_O < 150
		THEN
		PilaK2_O:=PilaK2_O+1;
		ELSE
		PilaK2_O:=0;		
	END_IF
END_IF



IF NOT StopMyPilaStatus
	THEN
	StatusK2_O:= (PilaK2_O AND 16#FF)+ (StateK*256);// выдать свой статус в сеть в старшем байте и пилу в младшем байте
END_IF



IF NOT StopMyPilaReady
	THEN
	ReadyK2_O:= (PilaK2_O AND 16#FF)+ (ReadyK*256);// выдать свою готовность в сеть в старшем байте и пилу в младшем байте
END_IF

{IF defined (Use_MyCOM_in_Rezerv) }
{ELSE}
	// выдать в COM-rezerv in RWH-driver				
	%QW16:=PilaK2_O;
	%QW17:=StatusK2_O;
	%QW18:=ReadyK2_O;
{END_IF}

///////////////////////////////////////////////////////////////////////////////////////////////////
// Контроль пил для фиксации отключения контроллера - нет пилы Net и нет пилы COM одновременно
	Tst1Both(Pila:=PilaK1_O, TimeOut:=Timeout_NoPila_FromNetBoth, NoPila=>NoPila_FromNetBoth);
{IF defined (Use_MyCOM_in_Rezerv) }
		// для использования с моим COM-портом !!!
	Tst2Both(Pila:=COM202_PRG.PilaFromK1, TimeOut:=Timeout_NoPila_FromCOMBoth, NoPila=>NoPila_FromCOMBoth);
{ELSE}
	Tst2Both(Pila:=%IW16, TimeOut:=Timeout_NoPila_FromCOMBoth, NoPila=>NoPila_FromCOMBoth);
{END_IF}
///////////////////////////////////////////////////////////////////////////////////////////////////


///////////////////////////////////////////////////////////////////////////////////////////////////
// Контроль пил для переключения каналов резервирования: Net - COM
	Tst1(Pila:=PilaK1_O, TimeOut:=Timeout_NoPila_FromNet, NoPila=>NoPila_FromNet);
{IF defined (Use_MyCOM_in_Rezerv) }
		// для использования с моим COM-портом !!!
	Tst2(Pila:=COM202_PRG.PilaFromK1, TimeOut:=Timeout_NoPila_FromCOM, NoPila=>NoPila_FromCOM);
{ELSE}
	Tst2(Pila:=%IW16, TimeOut:=Timeout_NoPila_FromCOM, NoPila=>NoPila_FromCOM);
{END_IF}
///////////////////////////////////////////////////////////////////////////////////////////////////


	IF NOT NoPila_FromNet
		THEN//есть пила по NET - работаем по сети
		REZZ1(_BMPERR:={BMPERR2}BMPERR_I, _My_MX_Status:={My_MX_Status}MxStatus_I, 
				_PilaK_O:= PilaK1_O, _StatusK_O:=StatusK1_O, _ReadyK_O:=ReadyK1_O,
				 _NumK:=2,// это контроллер №2
					_StateK:=StateK, _ReadyK:=ReadyK, _Cmd_GoPassive:=Cmd_GoPassive,
					_NoPilaBoth:=NoPila_FromCOMBoth AND NoPila_FromNetBoth AND (MxStatus_I.15),// 02 ноя 2012
					_NoPilaCommon=>NoPila_FromREZ, 
					_My_MX_Mode=>{My_MX_Mode}{%QW1}MxMode_O, _Udo=>My_Udo, _MasterOPC=>MasterOPC, _StateStr=>StateStr, _ReadyStr=>ReadyStr);
		
		ELSE//нет пилы по NET - работаем по СОМ
{IF defined (Use_MyCOM_in_Rezerv) }
		// для использования с моим COM-портом !!!
		// 	сделать задачи TaskCOM (запускает COM102_PRG), TaskCOM101(запускает COM101_PRG) в К1
		//     и задачи TaskCOM(запускает COM202_PRG), TaskCOM201(запускает COM201_PRG) в К2
		REZZ1(_BMPERR:={BMPERR2}BMPERR_I, _My_MX_Status:={My_MX_Status}MxStatus_I,
				_PilaK_O:= COM202_PRG.PilaFromK1, _StatusK_O:= COM202_PRG.StatusFromK1, _ReadyK_O:= COM202_PRG.ReadyFromK1,
				 _NumK:=2,// это контроллер №2
					_StateK:=StateK, _ReadyK:=ReadyK, _Cmd_GoPassive:=Cmd_GoPassive,
					_NoPilaBoth:=NoPila_FromCOMBoth AND NoPila_FromNetBoth AND (MxStatus_I.15),// 02 ноя 2012
					_NoPilaCommon=>NoPila_FromREZ, 
					_My_MX_Mode=>{My_MX_Mode}{%QW1}MxMode_O, _Udo=>My_Udo, _MasterOPC=>MasterOPC, _StateStr=>StateStr, _ReadyStr=>ReadyStr);
{ELSE}
		REZZ1(_BMPERR:={BMPERR2}BMPERR_I, _My_MX_Status:={My_MX_Status}MxStatus_I,
				_PilaK_O:= %IW16, _StatusK_O:= %IW17, _ReadyK_O:= %IW18,
				 _NumK:=2,// это контроллер №2
					_StateK:=StateK, _ReadyK:=ReadyK, _Cmd_GoPassive:=Cmd_GoPassive,
					_NoPilaBoth:=NoPila_FromCOMBoth AND NoPila_FromNetBoth AND (MxStatus_I.15),// 02 ноя 2012
					_NoPilaCommon=>NoPila_FromREZ, 
					_My_MX_Mode=>{My_MX_Mode}{%QW1}MxMode_O, _Udo=>My_Udo, _MasterOPC=>MasterOPC, _StateStr=>StateStr, _ReadyStr=>ReadyStr);
{END_IF}
	END_IF


//////// добавлено вместо закомментированого 8 апр 2013//////исправляем включение другого К ///////////////////////////
{IF defined (Use_U24Imp_in_Rezerv) }
// импульсное управление Udo	

	{IF defined (Use_U24ImpNotOnlySingleMode_in_Rezerv) }
	// импульсное управление Udo в режимах Active и Passive, но потенциальное удержание в Single	
		IF (StateK=Active)OR(StateK=Passive)
			THEN
			TP_Udo(in:=My_Udo, pt:=Imp_U24, Q=>Udo);
		END_IF
		IF (StateK=Single)
			THEN
			Udo:=My_Udo;	
		END_IF
	{ELSE}
			TP_Udo(in:=My_Udo, pt:=Imp_U24, Q=>Udo);
	{END_IF}

	{IF defined (Use_U24ImpRedire_in_Rezerv) }	
	// Периодический импульс подтверждения установки реле питания +24В в режимах Active/Single (добавлено 9 апр 2013)
	IF (StateK=Active)OR(StateK=Single)
		THEN
		IF (Redire_Udo_Cnt < Redire_Udo_CntMax)
			THEN
				Redire_Udo_Cnt:=Redire_Udo_Cnt+1;
			ELSE
				Redire_Udo_Cnt:=0;
				Udo:=1;
		END_IF
	END_IF
	{END_IF}
	
	{IF defined (Use_U24ImpOnStart_in_Rezerv)}
	// Импульс для подавления паразитного переключения Udo при включении другого контроллера
	IF (StateK=Active)OR(StateK=Single)
		THEN
		TP2_Udo(in:=DI_K[{11}9].RR.0, pt:=ImpLong_U24);
		IF TP2_Udo.Q
			THEN
			Udo:=1;
		END_IF
	END_IF
	{END_IF}

{ELSE}
// без импульса - потенциальное управление Udo	
	Udo:=My_Udo;	
{END_IF}
//////// окончание добавленого вместо закомментированого 8 апр 2013//////исправляем включение другого К ///////////////

	// в Помарской не прописан Udo прямо во вкладке DO поз.4 (как в ГавЯм DO_bit3 поз.16) - Фалеев 29.05.2018
	DO_K[3].RR.3:=	Udo;// подать напр на выходы	

	// в Помарской пилу активности для меандра
	//StopMyPilaAktiv  :=	NOT ((StateK=Single)OR(StateK=Active));// остановить пилу только в пассиве
	StopMyPilaAktiv  :=	((StateK=Active)AND((ReadyK1_O AND 16#FF00)=0)AND(BMPERR_I.7)) OR	// Я активный, другой (K1) не готов и у меня есть ошибка АВ УСО (поз8) - остановить пилу АКТ.
						((StateK=Single)AND (BMPERR_I.7)) OR				// Я один и у меня есть ошибка АВ УСО (поз8) - остановить пилу АКТ.
						(StateK=Passive)OR(StateK=Nothing);					// Я пассивный или ничего - остановить пилу АКТ.
	
	// формировать пилу активности для меандра акт DO
	IF NOT StopMyPilaAktiv
		THEN
			PilaAktiv:=PilaAktiv+1;
	END_IF
	DO_K[3].RR.0:=	PilaAktiv.0;	// вывести в DO3_bit0	 меандр активности   поз.4
	//DO_K[3].RR.11:=	PilaAktiv.0;	// вывести в DO3_bit11	 (для К1 индикация на дверь)   поз.4
	DO_K[3].RR.12:=	PilaAktiv.0;	// вывести в DO3_bit12	 (для К2 индикация на дверь)   поз.4


// просто индикация для   ПОМАРСКОЙ   !!!
	DO_K[2].RR.8:=NoPila_FromNet;
	DO_K[2].RR.9:=NoPila_FromCOM;
	DO_K[2].RR.11:=Udo;// подать напр на выходы	
	DO_K[2].RR.13:=(BMPERR_I <> 0);
	DO_K[2].RR.15:=NoPila_FromREZ;

	CASE StateK OF
 	Single:
			DO_K[2].RR.10:= 1;// Single
			DO_K[2].RR.12:= 0;// Active
			DO_K[2].RR.14:= 0;// Passive

	Active:	
			DO_K[2].RR.10:= 0;// Single
			DO_K[2].RR.12:= 1;// Active
			DO_K[2].RR.14:= 0;// Passive
	
	Passive:
			DO_K[2].RR.10:= 0;// Single
			DO_K[2].RR.12:= 0;// Active
			DO_K[2].RR.14:= 1;// Passive
	
	END_CASE	
	
	
END_CASE

END_PROGRAM

// REZERV1/PilaTst
FUNCTION_BLOCK PilaTst
VAR_INPUT
	Pila:WORD;
	TimeOut:TIME;
END_VAR
VAR_OUTPUT
	NoPila:BOOL;// нет пилы = True
END_VAR
VAR
	Pila_:WORD:=0;// значение пилы на предыдущем цикле
	T1:TON;
END_VAR

IF Pila=Pila_
	THEN
	T1.IN:=1;
//	T1.PT:=T#5000MS;
	T1.PT:=TimeOut;
	ELSE
	T1.IN:=0;
END_IF

T1();
NoPila:=T1.Q;
Pila_:=Pila;// сохранить для след цикла

END_FUNCTION_BLOCK

// REZERV1/REZ1
FUNCTION_BLOCK REZ1
VAR CONSTANT
	Timeout_StartOn:TIME:=T#3000MS;//T#10000MS;	
	Timeout_StartTo:TIME:=T#2000MS;//T#3000MS;	
	Timeout_NoPila_Rezerv:TIME:=T#1500MS;//T#3000MS;	
		DTimeout:TIME:=T#0MS;//T#500MS;	
 	Count_PassiveToActive_Other:INT:=15;
END_VAR
VAR_INPUT
	_BMPERR:WORD;// ошибки УСО этого контроллера
	_My_MX_Status:WORD;// входная переменная как MX_Status
	_PilaK_O:WORD;// глоб сетевая посылка из соседнего
	_StatusK_O:WORD;// глоб сетевая посылка из соседнего
	_ReadyK_O:WORD;// глоб сетевая посылка из соседнего
	_NumK:WORD;		// номер этого контроллера: 1 или 2
	_NoPilaBoth:BOOL;// нет пил по обоим каналам одновременно - другой контроллер отключился	
END_VAR
VAR_IN_OUT
	_StateK:RezervState;// Статус контроллера
	_ReadyK:WORD;// Готовность к управлению
	_Cmd_GoPassive:WORD;// команда "Стать пассивным" (от МПУ или из-вне)
END_VAR
VAR_OUTPUT
	_My_MX_Mode:WORD;// выходная переменная как MX_Mode
	_Udo:BOOL:=FALSE;// Вкл/откл U пит +24В на DO
	_MasterOPC:BOOL:=FALSE;// Мастер-переменная ОРС	
	_StateStr:STRING;
	_ReadyStr:WSTRING;
	_NoPilaCommon:BOOL;
END_VAR
VAR
	NoPila_Rezerv:BOOL;// признак отсутствия пилы соседа
	NoPilaStatus_Rezerv:BOOL;// признак отсутствия пилы Статуса соседа
	NoPilaReady_Rezerv:BOOL;// признак отсутствия пилы Готовность соседа
(*		NoCOMPila_Rezerv:BOOL;// признак отсутствия пилы соседа через СОМ
		NoCOMPilaStatus_Rezerv:BOOL;// признак отсутствия пилы Статуса соседа через СОМ
		NoCOMPilaReady_Rezerv:BOOL;// признак отсутствия пилы Готовность соседа через СОМ   *)

	Tst1:PilaTst;// функц-блок наличия пилы соседа	
	SetState:SetStateK;// функц-блок установки статуса контролллера	
	PilaStat1:PilaStat;// функц-блок наличия пилы Статуса соседа и самого Статуса
	StatusK_OO:WORD;//статус, выделенный из ПилыСтатуса
	PilaReady1:PilaReady;// функц-блок наличия пилы Готовности соседа и самой Готовности
	ReadyK_OO:WORD;//готовность, выделенная из ПилыГотов

(*	Tst2:PilaTst;// функц-блок наличия пилы соседа через СОМ	
//	SetState:SetStateK;// функц-блок установки статуса контролллера	
	PilaStat2:PilaStat;// функц-блок наличия пилы Статуса соседа и самого Статуса через СОМ
	StatusK_OOO:WORD;//статус, выделенный из ПилыСтатуса через СОМ
	PilaReady2:PilaReady;// функц-блок наличия пилы Готовности соседа и самой Готовности через СОМ
	ReadyK_OOO:WORD;//готовность, выделенная из ПилыГотов через СОМ   *)
	
	TT1, TT2:TON;
	Cnt_PassiveToActive_Other:INT:=0;

END_VAR

// включить обработку мультиплексора в системе резервирования
{define Use_MX_in_Rezerv}
// отключить обработку мультиплексора в системе резервирования
//{undefine Use_MX_in_Rezerv}

// выдать в окно "Message" подсказку о наличие или отсутствии МХ в проекте и на контроллере
{IF defined (Use_MX_in_Rezerv) }
{info 'MX is present in ELPK'}
{ELSE}
{info 'MX is NOT present in ELPK'}
{END_IF}

CASE _StateK OF
0: _StateStr:='Nothing';
1: _StateStr:='Single';
2: _StateStr:='Active';
3: _StateStr:='Passive';
END_CASE

CASE _ReadyK OF
0: _ReadyStr:="НЕ готов к управлению";
1: _ReadyStr:="Готов к управлению";
END_CASE

IF _BMPERR <> 0
	THEN// есть ошибки УСО - сбросить мою готовность взять управление
	_ReadyK := 0;
	ELSE// нет ошибок УСО - установить мою готовность взять управление
	_ReadyK := 1;
END_IF

// задержка на старте - ничего не делать, пока не отработал таймер
TT1(IN:=1, PT:=Timeout_StartOn);
IF TT1.Q
	THEN
	// исполняется на старте пока таймер НЕ отработал
	TT2(IN:=1, PT:=Timeout_StartTo);
	IF (TT2.Q=TRUE) OR (_StateK <> Nothing) 
		THEN
		//
		ELSE	
		Tst1(Pila:=_PilaK_O, TimeOut:=Timeout_NoPila_Rezerv, NoPila=>NoPila_Rezerv);
		PilaStat1(PilaStatus:=_StatusK_O, TimeOut:=Timeout_NoPila_Rezerv-DTimeout, NoPila=>NoPilaStatus_Rezerv, MyStatus=>StatusK_OO);
		PilaReady1(PilaReady:=_ReadyK_O, TimeOut:=Timeout_NoPila_Rezerv, NoPila=>NoPilaReady_Rezerv, MyReady=>ReadyK_OO);

		IF NoPila_Rezerv OR NoPilaStatus_Rezerv OR NoPilaReady_Rezerv
			THEN
			// нет пилы соседа
{IF defined (Use_MX_in_Rezerv) }
			// MX есть в контроллере - тогда проверяем
			// если есть 8000 (т.е. сосед отпустил МХ или его нет), то можно установить режим SINGLE
			IF _My_MX_Status.15 = 1
				THEN
//				IF (_My_MX_Status AND 16#F)= 4
//					THEN
					SetState(MyState:=Single, StateK=> _StateK, Udo=> _Udo, MasterOPC=> _MasterOPC);
//				END_IF
				ELSE
				// если нет 8000 (т.е. сосед есть и он активен), то выбираем режим
					CASE (_My_MX_Status AND 16#F) OF
					4:	SetState(MyState:=Passive, StateK=> _StateK, Udo=> _Udo, MasterOPC=> _MasterOPC);
					8:	SetState(MyState:=Active, StateK=> _StateK, Udo=> _Udo, MasterOPC=> _MasterOPC);
					ELSE
						SetState(MyState:=Single, StateK=> _StateK, Udo=> _Udo, MasterOPC=> _MasterOPC);
					END_CASE
			END_IF
{ELSE}
		// MX нет в контроллере - тогда просто установить режим SINGLE
			SetState(MyState:=Single, StateK=> _StateK, Udo=> _Udo, MasterOPC=> _MasterOPC);
{END_IF}
///			SetState(MyState:=Single, StateK=> _StateK, Udo=> _Udo, MasterOPC=> _MasterOPC);
			ELSE
			// есть пила соседа
			IF (StatusK_OO=Active) OR (StatusK_OO=Single)
				THEN
				SetState(MyState:=Passive, StateK=> _StateK, Udo=> _Udo, MasterOPC=> _MasterOPC);
				ELSE
				SetState(MyState:=Active, StateK=> _StateK, Udo=> _Udo, MasterOPC=> _MasterOPC);
			END_IF
		END_IF
	END_IF
	ELSE
	// пока задержка на старте - контролировать пилу, чтобы таймаут вышел (если нет связи)
	Tst1(Pila:=_PilaK_O, TimeOut:=Timeout_NoPila_Rezerv, NoPila=>NoPila_Rezerv);	
	PilaStat1(PilaStatus:=_StatusK_O, TimeOut:=Timeout_NoPila_Rezerv-DTimeout, NoPila=>NoPilaStatus_Rezerv, MyStatus=>StatusK_OO);
	PilaReady1(PilaReady:=_ReadyK_O, TimeOut:=Timeout_NoPila_Rezerv, NoPila=>NoPilaReady_Rezerv, MyReady=>ReadyK_OO);
END_IF

/////////////////   РАБОТА   //////////////////////////////////////////////////////
CASE _StateK OF
Nothing:
Single:	
	Tst1(Pila:=_PilaK_O, TimeOut:=Timeout_NoPila_Rezerv, NoPila=>NoPila_Rezerv);
	PilaStat1(PilaStatus:=_StatusK_O, TimeOut:=Timeout_NoPila_Rezerv-DTimeout, NoPila=>NoPilaStatus_Rezerv, MyStatus=>StatusK_OO);
	PilaReady1(PilaReady:=_ReadyK_O, TimeOut:=Timeout_NoPila_Rezerv, NoPila=>NoPilaReady_Rezerv, MyReady=>ReadyK_OO);

////	IF NoPila_Rezerv OR NoPilaStatus_Rezerv OR NoPilaReady_Rezerv
/////	IF NoPilaStatus_Rezerv	// отказ определять только по пиле статуса !!!
	IF NoPilaStatus_Rezerv OR _NoPilaBoth	// отказ определять по пиле статуса и при отсут обоих пил наверху
		THEN
		// нет пилы соседа
		SetState(MyState:=Single, StateK=> _StateK, Udo=> _Udo, MasterOPC=> _MasterOPC);
		ELSE
		// есть пила соседа
		IF (StatusK_OO=Passive)
			THEN
			SetState(MyState:=Active, StateK=> _StateK, Udo=> _Udo, MasterOPC=> _MasterOPC);
			ELSIF (StatusK_OO=Active) OR (StatusK_OO=Single)
				THEN	
				SetState(MyState:=Passive, StateK=> _StateK, Udo=> _Udo, MasterOPC=> _MasterOPC);
		END_IF
	END_IF
	_Cmd_GoPassive:=0;//сбросить возможную команду - не должно быть в Single
	{IF defined (Use_MX_in_Rezerv) }
	// если есть 8000 (т.е. сосед отпустил МХ), то можно делать МХ активным
	IF _My_MX_Status.15 = 1
		THEN
		_My_MX_Mode:=8;		
	END_IF
	{END_IF}

Active:
	Tst1(Pila:=_PilaK_O, TimeOut:=Timeout_NoPila_Rezerv, NoPila=>NoPila_Rezerv);
	PilaStat1(PilaStatus:=_StatusK_O, TimeOut:=Timeout_NoPila_Rezerv, NoPila=>NoPilaStatus_Rezerv, MyStatus=>StatusK_OO);
	PilaReady1(PilaReady:=_ReadyK_O, TimeOut:=Timeout_NoPila_Rezerv-DTimeout, NoPila=>NoPilaReady_Rezerv, MyReady=>ReadyK_OO);

////	IF NoPila_Rezerv OR NoPilaStatus_Rezerv OR NoPilaReady_Rezerv
/////	IF NoPilaReady_Rezerv	// отказ определять только по пиле готовности !!!
	IF NoPilaReady_Rezerv OR _NoPilaBoth	// отказ определять по пиле готовности и при отсут обоих пил наверху
		THEN
		// нет пилы соседа
		SetState(MyState:=Single, StateK=> _StateK, Udo=> _Udo, MasterOPC=> _MasterOPC);
		ELSE // есть пила соседа
		IF (StatusK_OO=Active)AND(_NumK=2)	// если сосед активен, а мой контроллер №2, то перейти в Пассив
			THEN
				SetState(MyState:=Passive, StateK=> _StateK, Udo=> _Udo, MasterOPC=> _MasterOPC);
///		IF ReadyK_OO = 1
			ELSIF (ReadyK_OO = 1)
			THEN// другой контроллер готов взять управление -  проверить мои ошибки УСО
			IF _BMPERR <> 0
				THEN// есть ошибки УСО - сбросить мой признак "Готов к управлению" и перейти в Passive
//				ReadyK := 0;
				Cnt_PassiveToActive_Other:= Count_PassiveToActive_Other{3};// 3 цикла ждать перехода соседа в Active, не реагируя на его статус
				SetState(MyState:=Passive, StateK=> _StateK, Udo=> _Udo, MasterOPC=> _MasterOPC);
				ELSE// нет ошибок УСО - установить мой признак "Готов к управлению" и проверить команду "Перейти в Пассив"
//				ReadyK := 1;
				IF _Cmd_GoPassive <> 0
					THEN// есть команда "Перейти в Пассив" - перейти в Passive
					_Cmd_GoPassive:=0;//сбросить команду
					Cnt_PassiveToActive_Other:= Count_PassiveToActive_Other{3};// 3 цикла ждать перехода соседа в Active, не реагируя на его статус
					SetState(MyState:=Passive, StateK=> _StateK, Udo=> _Udo, MasterOPC=> _MasterOPC);
					ELSE// нет команды "Перейти в Пассив" - остаться в Active
					SetState(MyState:=Active, StateK=> _StateK, Udo=> _Udo, MasterOPC=> _MasterOPC);
				END_IF
			END_IF
			ELSE// другой контроллер НЕ готов взять управление - остаться в Active
			SetState(MyState:=Active, StateK=> _StateK, Udo=> _Udo, MasterOPC=> _MasterOPC);
		END_IF
	END_IF
	{IF defined (Use_MX_in_Rezerv) }
	// если есть 8000 (т.е. сосед отпустил МХ), то можно делать МХ активным
	IF _My_MX_Status.15 = 1
		THEN
		_My_MX_Mode:=8;		
// начало добавления 30.10.12
		ELSE
		IF _My_MX_Status.3 = 1	// =8
			THEN
			_My_MX_Mode:=8;		
		END_IF
// конец добавления 30.10.12
	END_IF
	{END_IF}

Passive:
	Tst1(Pila:=_PilaK_O, TimeOut:=Timeout_NoPila_Rezerv, NoPila=>NoPila_Rezerv);
	PilaStat1(PilaStatus:=_StatusK_O, TimeOut:=Timeout_NoPila_Rezerv-DTimeout, NoPila=>NoPilaStatus_Rezerv, MyStatus=>StatusK_OO);
	PilaReady1(PilaReady:=_ReadyK_O, TimeOut:=Timeout_NoPila_Rezerv, NoPila=>NoPilaReady_Rezerv, MyReady=>ReadyK_OO);

///	IF NoPila_Rezerv OR NoPilaStatus_Rezerv OR NoPilaReady_Rezerv
///		THEN
///		// нет пилы соседа
///		SetState(MyState:=Single, StateK=> _StateK, Udo=> _Udo, MasterOPC=> _MasterOPC);
////	IF NoPila_Rezerv OR NoPilaStatus_Rezerv OR NoPilaReady_Rezerv
/////	IF NoPilaStatus_Rezerv	// отказ определять только по пиле статуса !!!
	IF NoPilaStatus_Rezerv OR _NoPilaBoth	// отказ определять по пиле статуса и при отсут обоих пил наверху
		THEN
		// нет пилы соседа
		{IF defined (Use_MX_in_Rezerv) }
		// MX есть в контроллере - тогда проверяем
		// если есть 8004 (т.е. сосед отпустил МХ или его нет, а я пассивный), то можно установить режим SINGLE
		IF _My_MX_Status = 16#8004
			THEN
			SetState(MyState:=Single, StateK=> _StateK, Udo=> _Udo, MasterOPC=> _MasterOPC);
		END_IF
		{ELSE}
		// MX нет в контроллере - тогда просто установить режим SINGLE
			SetState(MyState:=Single, StateK=> _StateK, Udo=> _Udo, MasterOPC=> _MasterOPC);
		{END_IF}
		ELSE
		// есть пила соседа
(*		IF (StatusK_OO = Nothing)
			THEN
				EXIT;// не делать ничего - оставить режим как есть !!!
			END_IF *)
		IF (StatusK_OO = Active) OR (StatusK_OO = Single)
			THEN
//			IF BMPERR1 <> 0
//				THEN// есть ошибки УСО - сбросить мою готовность взять управление
//				ReadyK := 0;
//				ELSE// нет ошибок УСО - установить мою готовность взять управление
//				ReadyK := 1;
//			END_IF
			SetState(MyState:=Passive, StateK=> _StateK, Udo=> _Udo, MasterOPC=> _MasterOPC);
			Cnt_PassiveToActive_Other:= 0;
			ELSIF (StatusK_OO = Nothing)
				THEN// если статус соседа = 0, то не делать ничего - оставить режим как есть !!!
				//
			ELSE
			IF Cnt_PassiveToActive_Other <= 0
				THEN// не надо задержек в реакции
				// сосед не в Active - перейти в Active мне
				SetState(MyState:=Active, StateK=> _StateK, Udo=> _Udo, MasterOPC=> _MasterOPC);
				ELSE
				// счетчик > 0 - только что был переход меня из А в Р - надо ждать пока сосед изменит статус !!!	
				// ждем несколько циклов
				Cnt_PassiveToActive_Other:=Cnt_PassiveToActive_Other-1;
			END_IF
		END_IF
	END_IF
	_Cmd_GoPassive:=0;//сбросить возможную команду - не должно быть в Passive
	{IF defined (Use_MX_in_Rezerv) }
	_My_MX_Mode:=4;
	{END_IF}
	
END_CASE
//
// Посылать команду в отладочном проекте из визуализации надо в переменную Cmd_GoPassive в виде одной из 1 в слове
//
// Суммарный признак отсутствия связи по трем пилам - поднять наверх
_NoPilaCommon:= NoPila_Rezerv OR NoPilaStatus_Rezerv OR NoPilaReady_Rezerv;

END_FUNCTION_BLOCK

// REZERV1/PilaReady
FUNCTION_BLOCK PilaReady
VAR_INPUT
	PilaReady:WORD;
	TimeOut:TIME;
END_VAR
VAR_OUTPUT
	NoPila:BOOL;// нет пилы = True
	MyReady:WORD;	
END_VAR
VAR
	Pila:WORD:=0;// значение пилы на текущем цикле
	Pila_:WORD:=0;// значение пилы на предыдущем цикле
	T1:TON;
END_VAR

MyReady:= SHR( PilaReady,8) AND 16#FF;// готовность в ст байте
Pila:= PilaReady AND 16#FF;// пила в мл байте
IF Pila=Pila_
	THEN
	T1.IN:=1;
//	T1.PT:=T#5000MS;
	T1.PT:=TimeOut;
	ELSE
	T1.IN:=0;
END_IF

T1();
NoPila:=T1.Q;
IF T1.Q
	THEN
	MyReady:=0;
END_IF

Pila_:=Pila;// сохранить для след цикла

END_FUNCTION_BLOCK

// REZERV1/SetStateK
FUNCTION_BLOCK SetStateK
VAR_INPUT
	MyState:RezervState;
END_VAR
VAR_OUTPUT
	StateK:RezervState;
	Udo:BOOL;
	MasterOPC:BOOL;
END_VAR
VAR
END_VAR

CASE MyState OF
Nothing:

Single:	
		StateK:=RezervState.Single;//установить статус контроллера Single
		Udo:=TRUE;//включить питание DO 
		MasterOPC:=TRUE;// передавать в ОРС с этого контроллера

Active:
		StateK:=RezervState.Active;//установить статус контроллера Active
		Udo:=TRUE;//включить питание DO 
		MasterOPC:=TRUE;// передавать в ОРС с этого контроллера

Passive:	
		StateK:=RezervState.Passive;//установить статус контроллера Passive
		Udo:=FALSE;//отключить питание DO 
		MasterOPC:=FALSE;// НЕ передавать в ОРС с этого контроллера

END_CASE

END_FUNCTION_BLOCK

// REZERV1/PilaStat
FUNCTION_BLOCK PilaStat
VAR_INPUT
	PilaStatus:WORD;
	TimeOut:TIME;
END_VAR
VAR_OUTPUT
	NoPila:BOOL;// нет пилы = True
	MyStatus:WORD;	
END_VAR
VAR
	Pila:WORD:=0;// значение пилы на текущем цикле
	Pila_:WORD:=0;// значение пилы на предыдущем цикле
	T1:TON;
END_VAR

MyStatus:= SHR( PilaStatus,8) AND 16#FF;// статус в ст байте
Pila:= PilaStatus AND 16#FF;// пила в мл байте
IF Pila=Pila_
	THEN
	T1.IN:=1;
//	T1.PT:=T#5000MS;
	T1.PT:=TimeOut;
	ELSE
	T1.IN:=0;
END_IF

T1();
NoPila:=T1.Q;
IF T1.Q
	THEN
	MyStatus:=0;
END_IF

Pila_:=Pila;// сохранить для след цикла

END_FUNCTION_BLOCK

// lowLevel_ecl/kontroller/execKontrollersInputs
FUNCTION execKontrollersInputs : bool
VAR_INPUT
	CONSTANT table:TableDescriptor;
END_VAR
VAR
	curObject:POINTER TO BaseObject;
	curKontroller:IKontroller;
END_VAR

curObject:=table.head;
IF curObject=0 THEN
	RETURN;
END_IF
REPEAT
	IF (__QUERYINTERFACE(curObject^,curKontroller)) THEN		
		curKontroller.callInputTable();
	END_IF;
	curObject:=curObject^.getNext();
	UNTIL curObject=0
END_REPEAT

END_FUNCTION

// lowLevel_ecl/kontroller/execKontrollersOutputs
FUNCTION execKontrollersOutputs : bool
VAR_INPUT
	CONSTANT table:TableDescriptor;
END_VAR
VAR
	curObject:POINTER TO BaseObject;
	curKontroller:IKontroller;
END_VAR

curObject:=table.head;
IF curObject=0 THEN
	RETURN;
END_IF
REPEAT
	IF (__QUERYINTERFACE(curObject^,curKontroller)) THEN		
		curKontroller.callOutputTable();
	END_IF;
	curObject:=curObject^.getNext();
	UNTIL curObject=0
END_REPEAT

END_FUNCTION

// Elpk_03_02_COMMON/ELPK03_to_MLP_OUT
PROGRAM ELPK03_to_MLP_OUT
VAR_INPUT
	DO2_BLK: WORD;
	DO3_BLK: WORD;
END_VAR
VAR
	I:INT;
END_VAR



(*
											//	s_Aux	:	WORD	;	//	bit-0 присутствие 1-есть, 0 -нет (привязка в конфигурации MLP)
																		//	bit-1 тип модуля 1-выходной, 0 -входной
																		//	bit-2 достоверность 1- достоверно,0- не достоверно
									  		//	kcc		:	WORD	;   //	Контроль Целостности Цепи - КЦЦ
																		//	каждая цепь 2 бита
																		//	00 - неизвестно или обрыв цепи
																		//	01 - есть Целостность Цепи
																		//	10 - есть ток
																		//	11 - КЗ
											//	kk		:	WORD	;	//	Контроль выхода команды - КК
																		//	каждая цепь 2 бита
																		//	00 - не бывает
																		//	01 - пассивное состояние
																		//	10 - активное (есть выход)состояние
																		//	11 - ошибка выхода команды 
									  		//	value_cc:	WORD	;	//	содержимое выходных регистров 
	*)
	
	
	
	//	
	//kontroller.Din_Dout[0].s_Aux		:= 7;	// .0 - есть в проекте		.1 - входные		.2 - достоверность		
	//kontroller.Din_Dout[0].s_Aux.2		:= DO_K[0].VeraB;	// достоверность из драйвера RWH (=1 - достоверно)	
	//kontroller.Din_Dout[0].s_Aux.2		:= (kontroller.DIn_Dout[0].value_cc.1=0);		// недостоверность - получим их NodeErr модуля ???		
	//
	//kontroller.Din_Dout[0].kcc.0		:= 1;	// 01 - есть Целостность цепи 		
	//kontroller.Din_Dout[0].kcc.1		:= 0;	// 01 - есть Целостность цепи 		
	//kontroller.Din_Dout[0].kk.0		:= 0;	// 01 - пассивное состояние			 10 - активное состояние 		
	//kontroller.Din_Dout[0].kk.1		:= 1;	// 01 - пассивное состояние			 10 - активное состояние 		
	// 01 - пассивное состояние			 10 - активное состояние 		
	//kontroller.Din_Dout[0].kk.0	:=	NOT kontroller.Dout_[0].0;// 01 - пассивное состояние			 10 - активное состояние
	//kontroller.Din_Dout[0].kk.1	:=	    kontroller.Dout_[0].0;// 01 - пассивное состояние			 10 - активное состояние

	//kontroller.Din_Dout[0].value_cc	:= kontroller.Dout_[0];	//	содержимое выходных регистров		
					

	//***********************************************************************************************************************************************************************
	//
	//	если нет обращений в программе к	std12k5.DO_K[].Q или нет питания +24В	, то Vera.0=FALSE,
	//	если программа обращается к 	std12k5.DO_K[].Q и есть питание +24В	, то Vera.0=TRUE
	//		остальные биты Vera всегда = FALSE
	//
	//***********************************************************************************************************************************************************************
	//	DOUT	поз.2
	DO_K[2].VeraB:=	DO_K[2].Vera.0; 
	//	DOUT	поз.4
	DO_K[3].VeraB:=	DO_K[3].Vera.0; 
	//	DOUT	поз.5
	DO_K[0].VeraB:=	DO_K[0].Vera.0; 
	//	DOUT	поз.6
	DO_K[4].VeraB:=	DO_K[4].Vera.0; 
	//	DOUT	поз.7
	DO_K[1].VeraB:=	DO_K[1].Vera.0; 
	


//	ЭЛПК-03-02   МТЦ03-16-Ш (поз.5)											 
	DO_K[0].RR.0:=	kontroller.Dout_[0].0;	// Кран 1 открыть
	DO_K[0].RR.1:=	kontroller.Dout_[0].1;	// Кран 1 закрыть (есть в БЭАО)
	DO_K[0].RR.2:=	kontroller.Dout_[0].2;	// Кран 2 открыть
	DO_K[0].RR.3:=	kontroller.Dout_[0].3;	// Кран 2 закрыть (есть в БЭАО)
	DO_K[0].RR.4:=	kontroller.Dout_[0].4;	// Кран 3 открыть
	DO_K[0].RR.5:=	kontroller.Dout_[0].5;	// Кран 3 закрыть (есть в БЭАО)
	DO_K[0].RR.6:=	kontroller.Dout_[0].6;	// Кран 3бис открыть (есть в БЭАО)
	DO_K[0].RR.7:=	kontroller.Dout_[0].7;	// Кран 3бис закрыть
	DO_K[0].RR.8:=	kontroller.Dout_[0].8;	// Кран 4 открыть
	DO_K[0].RR.9:=	kontroller.Dout_[0].9;	// Кран 4 закрыть (есть в БЭАО)
	DO_K[0].RR.10:=	kontroller.Dout_[0].10;	// Кран 5 открыть (есть в БЭАО, можно таймер)
	DO_K[0].RR.11:=	kontroller.Dout_[0].11;	// Кран 5 закрыть
	DO_K[0].RR.12:=	kontroller.Dout_[0].12;	// Кран 6 открыть (есть в БЭАО)
	DO_K[0].RR.13:=	kontroller.Dout_[0].13;	// Кран 6 закрыть
	DO_K[0].RR.14:=	kontroller.Dout_[0].14;	// Смазку крана 1 включить
	DO_K[0].RR.15:=	kontroller.Dout_[0].15;	// Смазку крана 2 включить
		//	
		kontroller.Din_Dout[0].s_Aux		:= 7;	// .0 - есть в проекте		.1 - входные		.2 - достоверность		
		kontroller.Din_Dout[0].s_Aux.2		:= DO_K[0].VeraB;	// достоверность из драйвера RWH (=1 - достоверно)	
		//kontroller.Din_Dout[0].s_Aux.2		:= (kontroller.DIn_Dout[0].value_cc.1=0);		// недостоверность - получим их NodeErr модуля ???		
		DO_03_kk(K_Dout:= kontroller.Dout_[0], K_Din_Dout_kk:= kontroller.Din_Dout[0]);		// добавить диагностику выходов
		//

//	ЭЛПК-03-02   МТЦ03-16-Ш (поз.7)											 
	DO_K[1].RR.0:=	kontroller.Dout_[1].0;	// Включить ПНС (есть в БЭАО)
	DO_K[1].RR.1:=	kontroller.Dout_[1].1;	// Отключить ПНС
	DO_K[1].RR.2:=	kontroller.Dout_[1].2;	// резерв
	DO_K[1].RR.3:=	kontroller.Dout_[1].3;	// резерв
	DO_K[1].RR.4:=	kontroller.Dout_[1].4;	// Включить НУ1
	DO_K[1].RR.5:=	kontroller.Dout_[1].5;	// Отключить НУ1
	DO_K[1].RR.6:=	kontroller.Dout_[1].6;	// Включить НУ2
	DO_K[1].RR.7:=	kontroller.Dout_[1].7;	// Отключить НУ2
	DO_K[1].RR.8:=	kontroller.Dout_[1].8;	// Включить вентилятор АВОМ 1
	DO_K[1].RR.9:=	kontroller.Dout_[1].9;	// Отключить вентилятор АВОМ 1
	DO_K[1].RR.10:=	kontroller.Dout_[1].10;	// Включить вентилятор АВОМ 2
	DO_K[1].RR.11:=	kontroller.Dout_[1].11;	// Отключить вентилятор АВОМ 2
	DO_K[1].RR.12:=	kontroller.Dout_[1].12;	// Включить вентилятор АВОМ 3
	DO_K[1].RR.13:=	kontroller.Dout_[1].13;	// Отключить вентилятор АВОМ 3
	DO_K[1].RR.14:=	kontroller.Dout_[1].14;	// Включить вентилятор АВОМ 4
	DO_K[1].RR.15:=	kontroller.Dout_[1].15;	// Отключить вентилятор АВОМ 4
		//	
		kontroller.Din_Dout[1].s_Aux		:= 7;	// .0 - есть в проекте		.1 - входные		.2 - достоверность		
		kontroller.Din_Dout[1].s_Aux.2		:= DO_K[1].VeraB;	// достоверность из драйвера RWH (=1 - достоверно)	
		//kontroller.Din_Dout[1].s_Aux.2		:= (kontroller.DIn_Dout[1].value_cc.1=0);		// недостоверность - получим их NodeErr модуля ???		
		DO_03_kk(K_Dout:= kontroller.Dout_[1], K_Din_Dout_kk:= kontroller.Din_Dout[1]);		// добавить диагностику выходов
		//

//	ЭЛПК-03-02   МТЦ03-16-Ш (поз.2)											 
	DO_K[2].RR.0:=	kontroller.Dout_[2].0;	// Включить калорифер АВОМ
	DO_K[2].RR.1:=	kontroller.Dout_[2].1;	// Отключить калорифер АВОМ
	DO_K[2].RR.2:=	kontroller.Dout_[2].2;	// Включить ТЭН м/б
	DO_K[2].RR.3:=	kontroller.Dout_[2].3;	// Отключить ТЭН м/б
	DO_K[2].RR.4:=	kontroller.Dout_[2].4;	// Включить насос циркуляции масла в м/б
	DO_K[2].RR.5:=	kontroller.Dout_[2].5;	// Отключить насос циркуляции масла в м/б
	DO_K[2].RR.6:=	kontroller.Dout_[2].6;	// Включить электроподогрев колл. АВОМ
	DO_K[2].RR.7:=	kontroller.Dout_[2].7;	// Отключить электроподогрев колл. АВОМ
(*	DO_K[2].RR.8:=	kontroller.Dout_[2].8;	// резерв
	DO_K[2].RR.9:=	kontroller.Dout_[2].9;	// резерв
	DO_K[2].RR.10:=	kontroller.Dout_[2].10;	// резерв
	DO_K[2].RR.11:=	kontroller.Dout_[2].11;	// резерв
	DO_K[2].RR.12:=	kontroller.Dout_[2].12;	// резерв
	DO_K[2].RR.13:=	kontroller.Dout_[2].13;	// резерв
	DO_K[2].RR.14:=	kontroller.Dout_[2].14;	// резерв
	DO_K[2].RR.15:=	kontroller.Dout_[2].15;	// резерв   *)
	IF NOT DO2_BLK.8  THEN	DO_K[2].RR.8:=	kontroller.Dout_[2].8;	END_IF	// резерв
	IF NOT DO2_BLK.9  THEN	DO_K[2].RR.9:=	kontroller.Dout_[2].9;	END_IF	// резерв
	IF NOT DO2_BLK.10 THEN	DO_K[2].RR.10:=	kontroller.Dout_[2].10;	END_IF	// резерв
	IF NOT DO2_BLK.11 THEN	DO_K[2].RR.11:=	kontroller.Dout_[2].11;	END_IF	// резерв
	IF NOT DO2_BLK.12 THEN	DO_K[2].RR.12:=	kontroller.Dout_[2].12;	END_IF	// резерв
	IF NOT DO2_BLK.13 THEN	DO_K[2].RR.13:=	kontroller.Dout_[2].13;	END_IF	// резерв
	IF NOT DO2_BLK.14 THEN	DO_K[2].RR.14:=	kontroller.Dout_[2].14;	END_IF	// резерв
	IF NOT DO2_BLK.15 THEN	DO_K[2].RR.15:=	kontroller.Dout_[2].15;	END_IF	// резерв
		//	
		kontroller.Din_Dout[2].s_Aux		:= 7;	// .0 - есть в проекте		.1 - входные		.2 - достоверность		
		kontroller.Din_Dout[2].s_Aux.2		:= DO_K[2].VeraB;	// достоверность из драйвера RWH (=1 - достоверно)	
		//kontroller.Din_Dout[2].s_Aux.2		:= (kontroller.DIn_Dout[2].value_cc.1=0);		// недостоверность - получим их NodeErr модуля ???		
		DO_03_kk(K_Dout:= kontroller.Dout_[2], K_Din_Dout_kk:= kontroller.Din_Dout[2]);		// добавить диагностику выходов
		//
	
//	ЭЛПК-03-02   МТЦ03-16-Ш (поз.4)											 
(*	DO_K[3].RR.0:=	kontroller.Dout_[3].0;	// Для К1: Меандр активности К1						// Для К2: Меандр активности К2
	DO_K[3].RR.1:=	kontroller.Dout_[3].1;	// Для К1: Команда стать пассивным (от К1)			// Для К2: Команда стать пассивным (от К2)
	DO_K[3].RR.2:=	kontroller.Dout_[3].2;	// Для К1: Разрешить условный переход от К1			// Для К2: Разрешить условный переход от К2
	DO_K[3].RR.3:=	kontroller.Dout_[3].3;	// Для К1: Команда "Отключить выходы К2"			// Для К2: Команда "Отключить выходы К1"
	DO_K[3].RR.4:=	kontroller.Dout_[3].4;	// резерв
	DO_K[3].RR.5:=	kontroller.Dout_[3].5;	// резерв
	DO_K[3].RR.6:=	kontroller.Dout_[3].6;	// резерв
	DO_K[3].RR.7:=	kontroller.Dout_[3].7;	// резерв	*)
	IF NOT DO3_BLK.0  THEN	DO_K[3].RR.0:=	kontroller.Dout_[3].0;	END_IF	// Для К1: Меандр активности К1						// Для К2: Меандр активности К2
	IF NOT DO3_BLK.1  THEN	DO_K[3].RR.1:=	kontroller.Dout_[3].1;	END_IF	// Для К1: Команда стать пассивным (от К1)			// Для К2: Команда стать пассивным (от К2)
	IF NOT DO3_BLK.2  THEN	DO_K[3].RR.2:=	kontroller.Dout_[3].2;	END_IF	// Для К1: Разрешить условный переход от К1			// Для К2: Разрешить условный переход от К2
	IF NOT DO3_BLK.3  THEN	DO_K[3].RR.3:=	kontroller.Dout_[3].3;	END_IF	// Для К1: Команда "Отключить выходы К2"			// Для К2: Команда "Отключить выходы К1"
	IF NOT DO3_BLK.4  THEN	DO_K[3].RR.4:=	kontroller.Dout_[3].4;	END_IF	// резерв
	IF NOT DO3_BLK.5  THEN	DO_K[3].RR.5:=	kontroller.Dout_[3].5;	END_IF	// резерв
	IF NOT DO3_BLK.6  THEN	DO_K[3].RR.6:=	kontroller.Dout_[3].6;	END_IF	// резерв
	IF NOT DO3_BLK.7  THEN	DO_K[3].RR.7:=	kontroller.Dout_[3].7;	END_IF
	DO_K[3].RR.8:=	kontroller.Dout_[3].8;	// Индикация АС красный фонарь (фонарь + кнопка)
	DO_K[3].RR.9:=	kontroller.Dout_[3].9;	// Индикация ПС зеленый фонарь
	DO_K[3].RR.10:=	kontroller.Dout_[3].10;	// Индикация НО (подсветка кнопки на шкафу)
	(*DO_K[3].RR.11:=	kontroller.Dout_[3].11;	// К1 активен (зел.лампа на двери)*)
	IF NOT DO3_BLK.11  THEN	DO_K[3].RR.11:=	kontroller.Dout_[3].11;	END_IF	// К1 активен (зел.лампа на двери)
	(*DO_K[3].RR.12:=	kontroller.Dout_[3].12;	// К2 активен (зел.лампа на двери)*)
	IF NOT DO3_BLK.12  THEN	DO_K[3].RR.12:=	kontroller.Dout_[3].12;	END_IF	// К2 активен (зел.лампа на двери)
	DO_K[3].RR.13:=	kontroller.Dout_[3].13;	// Синхронизация режима ЭГПА (от К1)				// Синхронизация режима ЭГПА (от К2)
	DO_K[3].RR.14:=	kontroller.Dout_[3].14;	// резерв
	DO_K[3].RR.15:=	kontroller.Dout_[3].15;	// резерв
		//	
		kontroller.Din_Dout[3].s_Aux		:= 7;	// .0 - есть в проекте		.1 - входные		.2 - достоверность		
		kontroller.Din_Dout[3].s_Aux.2		:= DO_K[3].VeraB;	// достоверность из драйвера RWH (=1 - достоверно)	
		//kontroller.Din_Dout[3].s_Aux.2		:= (kontroller.DIn_Dout[3].value_cc.1=0);		// недостоверность - получим их NodeErr модуля ???		
		DO_03_kk(K_Dout:= kontroller.Dout_[3], K_Din_Dout_kk:= kontroller.Din_Dout[3]);		// добавить диагностику выходов
		//
		
//	ЭЛПК-03-02   МТЦ03-16-Ш (поз.6)											 
	DO_K[4].RR.0:=	kontroller.Dout_[4].0;	// Неисправность ГПА
	DO_K[4].RR.1:=	kontroller.Dout_[4].1;	// Авария ГПА (в ШКС-04М) (Есть в БЭАО)
	DO_K[4].RR.2:=	kontroller.Dout_[4].2;	// Работа ГПА (в ШКС-04М) (закрывает кран 6)
	DO_K[4].RR.3:=	kontroller.Dout_[4].3;	// Наличие напряжения =220В в ШУ (лампа на двери)
	DO_K[4].RR.4:=	kontroller.Dout_[4].4;	// резерв
	DO_K[4].RR.5:=	kontroller.Dout_[4].5;	// резерв
	DO_K[4].RR.6:=	kontroller.Dout_[4].6;	// Включить МВ
	DO_K[4].RR.7:=	kontroller.Dout_[4].7;	// Отключить МВ	(Есть в БЭАО)
	DO_K[4].RR.8:=	kontroller.Dout_[4].8;	// ПУСК
	DO_K[4].RR.9:=	kontroller.Dout_[4].9;	// ОСТАНОВ
	DO_K[4].RR.10:=	kontroller.Dout_[4].10;	// резерв
	DO_K[4].RR.11:=	kontroller.Dout_[4].11;	// резерв
	DO_K[4].RR.12:=	kontroller.Dout_[4].12;	// резерв
	DO_K[4].RR.13:=	kontroller.Dout_[4].13;	// резерв
	DO_K[4].RR.14:=	kontroller.Dout_[4].14;	// резерв
	DO_K[4].RR.15:=	kontroller.Dout_[4].15;	// резерв
		//	
		kontroller.Din_Dout[4].s_Aux		:= 7;	// .0 - есть в проекте		.1 - входные		.2 - достоверность		
		kontroller.Din_Dout[4].s_Aux.2		:= DO_K[4].VeraB;	// достоверность из драйвера RWH (=1 - достоверно)	
		//kontroller.Din_Dout[4].s_Aux.2		:= (kontroller.DIn_Dout[4].value_cc.1=0);		// недостоверность - получим их NodeErr модуля ???		
		DO_03_kk(K_Dout:= kontroller.Dout_[4], K_Din_Dout_kk:= kontroller.Din_Dout[4]);		// добавить диагностику выходов
		//
	
	
	
	
	
	

	FOR I:=0 TO 30 DO
		IF (Imitator_Code=16#55AA)
		THEN// имитатор вкл
			DO_K[I].Imx := Imitator_Code;
			DO_K[I].Im := DO_K[I].RR;	// в RR пишет прикладная программа!
			DO_K[I].VeraB := TRUE;
		ELSE
			DO_K[I].Imx := 0;
			DO_K[I].Q := DO_K[I].RR;	// в RR пишет прикладная программа!
		END_IF

		///DOs_Im[I]:= DO_K[I].Im;	// передать в имитатор	:	только для отладки моим имитатором !
	END_FOR

END_PROGRAM

// Elpk_03_02_COMMON/DO_03_kk
FUNCTION DO_03_kk : WORD
VAR_INPUT
	K_Dout:	WORD {BOOL};	
END_VAR
VAR_IN_OUT
	K_Din_Dout_kk: sDIN_DOUT; {WORD}
END_VAR
VAR
END_VAR

